# B&R Automation Studio project ABC_Pltzr
Automation Studio 4.2.4.149

## Configuration PPC70_24025GEN

### IoMap.iom - 4PPC70_101G_20W/IoMap.iom
```iecst
(*********************************************************************************
 * Copyright:
 * Author:    goran
 * Created:   August 31, 2015/10:10 PM
 *********************************************************************************
 * IO mapping
 *********************************************************************************)
VAR_CONFIG
	::gHWModules[1].ModuleOk AT %IX."X20BR9300".ModuleOk;
	::gHWModules[2].ModuleOk AT %IX."X20DI9371".ModuleOk;
	::gHWModules[3].ModuleOk AT %IX."X20DI9371a".ModuleOk;
	::gHWModules[4].ModuleOk AT %IX."X20DO4529".ModuleOk;
	::gHWModules[5].ModuleOk AT %IX."X20PS2100".ModuleOk;
	::gHWModules[6].ModuleOk AT %IX."X20DO9322".ModuleOk;
	gHWModules[7].ModuleOk AT %IX."X20DO9322a".ModuleOk;
	gHWModules[8].ModuleOk AT %IX."X20BT9400".ModuleOk;
	gHWModules[9].ModuleOk AT %IX."8I64-VFD1".ModuleOk;
	gHWModules[10].ModuleOk AT %IX."8I64-VFD2".ModuleOk;
	gHWModules[11].ModuleOk AT %IX."8I64-VFD5".ModuleOk;
	gHWModules[12].ModuleOk AT %IX."8I64-VFD52".ModuleOk;
	gHWModules[13].ModuleOk AT %IX."8I64-VFD11".ModuleOk;
	gHWModules[14].ModuleOk AT %IX."8I64-VFD12".ModuleOk;
	gHWModules[15].ModuleOk AT %IX."X67DM1321".ModuleOk;
	gHWModules[16].ModuleOk AT %IX."X67DM1321a".ModuleOk;
	gHWModules[17].ModuleOk AT %IX."X67DM1321.L08".ModuleOk;
	gHWModules[18].ModuleOk AT %IX."X67DM1321b".ModuleOk;
	::gMachineVFD[1].vfdIn.Status.ReadyToSwitchOn AT %IX."8I64-VFD1".ETAD_Input_Bool_00;
	::gMachineVFD[1].vfdIn.Status.SwitchedOn AT %IX."8I64-VFD1".ETAD_Input_Bool_01;
	::gMachineVFD[1].vfdIn.Status.OperationEnabled AT %IX."8I64-VFD1".ETAD_Input_Bool_02;
	::gMachineVFD[1].vfdIn.Status.FaultDetection AT %IX."8I64-VFD1".ETAD_Input_Bool_03;
	::gMachineVFD[1].vfdIn.Status.VoltageEnabled AT %IX."8I64-VFD1".ETAD_Input_Bool_04;
	::gMachineVFD[1].vfdIn.Status.QuickStop AT %IX."8I64-VFD1".ETAD_Input_Bool_05;
	::gMachineVFD[1].vfdIn.Status.SwitchOnDisabled AT %IX."8I64-VFD1".ETAD_Input_Bool_06;
	::gMachineVFD[1].vfdIn.Status.WarningAlarm AT %IX."8I64-VFD1".ETAD_Input_Bool_07;
	::gMachineVFD[1].vfdIn.Status.TargetReached AT %IX."8I64-VFD1".ETAD_Input_Bool_10;
	::gMachineVFD[1].vfdIn.Status.StopKey AT %IX."8I64-VFD1".ETAD_Input_Bool_14;
	::gMachineVFD[1].vfdIn.Status.Direction AT %IX."8I64-VFD1".ETAD_Input_Bool_15;
	::gMachineVFD[1].vfdIn.Status.Accelerating AT %IX."8I64-VFD1".ETI_Input_Bool_09;
	::gMachineVFD[1].vfdIn.Status.Decelerating AT %IX."8I64-VFD1".ETI_Input_Bool_10;
	::gMachineVFD[1].vfdIn.Status.FastStop AT %IX."8I64-VFD1".ETI_Input_Bool_12;
	::gMachineVFD[1].vfdIn.Status.CurrentVelocity AT %IW."8I64-VFD1".RFRD_Input;
	::gMachineVFD[1].vfdIn.Status.MotorTorque AT %IW."8I64-VFD1".OTR_Input;
	::gMachineVFD[1].vfdIn.Status.MotorCurrent AT %IW."8I64-VFD1".LCR_Input;
	::gMachineVFD[1].vfdIn.Status.DriveThermalState AT %IW."8I64-VFD1".THD_Input;
	::gMachineVFD[1].vfdIn.Status.MotorThermalState AT %IW."8I64-VFD1".THR_Input;
	::gMachineVFD[1].vfdIn.IO.LogicInput1 AT %IX."8I64-VFD1".IOLR_Input_Bool_00;
	::gMachineVFD[1].vfdIn.IO.LogicInput2 AT %IX."8I64-VFD1".IOLR_Input_Bool_01;
	::gMachineVFD[1].vfdIn.IO.LogicInput3 AT %IX."8I64-VFD1".IOLR_Input_Bool_02;
	::gMachineVFD[1].vfdIn.IO.LogicInput4 AT %IX."8I64-VFD1".IOLR_Input_Bool_03;
	::gMachineVFD[1].vfdIn.IO.Relay02State AT %IX."8I64-VFD1".IOLR_Input_Bool_09;
	::gMachineVFD[1].vfdIn.Fault.CurrentFault AT %IW."8I64-VFD1".ERRD_Input;
	::gMachineVFD[1].vfdIn.Fault.LastFault AT %IW."8I64-VFD1".LFT_Input;
	::gMachineVFD[1].vfdOut.Control.SwitchOn AT %QX."8I64-VFD1".CMDD_Output_Bool_00;
	::gMachineVFD[1].vfdOut.Control.DisableVoltage AT %QX."8I64-VFD1".CMDD_Output_Bool_01;
	::gMachineVFD[1].vfdOut.Control.QuickStop AT %QX."8I64-VFD1".CMDD_Output_Bool_02;
	::gMachineVFD[1].vfdOut.Control.EnableOperation AT %QX."8I64-VFD1".CMDD_Output_Bool_03;
	::gMachineVFD[1].vfdOut.Control.FaultReset AT %QX."8I64-VFD1".CMDD_Output_Bool_07;
	::gMachineVFD[1].vfdOut.Control.Direction AT %QX."8I64-VFD1".CMDD_Output_Bool_11;
	::gMachineVFD[1].vfdOut.Control.FastStop AT %QX."8I64-VFD1".CMDD_Output_Bool_12;
	::gMachineVFD[1].vfdOut.Control.VelocitySetpoint AT %QW."8I64-VFD1".LFRD_Output;
	::gMachineVFD[2].vfdIn.Status.ReadyToSwitchOn AT %IX."8I64-VFD2".ETAD_Input_Bool_00;
	::gMachineVFD[2].vfdIn.Status.SwitchedOn AT %IX."8I64-VFD2".ETAD_Input_Bool_01;
	::gMachineVFD[2].vfdIn.Status.OperationEnabled AT %IX."8I64-VFD2".ETAD_Input_Bool_02;
	::gMachineVFD[2].vfdIn.Status.FaultDetection AT %IX."8I64-VFD2".ETAD_Input_Bool_03;
	::gMachineVFD[2].vfdIn.Status.VoltageEnabled AT %IX."8I64-VFD2".ETAD_Input_Bool_04;
	::gMachineVFD[2].vfdIn.Status.QuickStop AT %IX."8I64-VFD2".ETAD_Input_Bool_05;
	::gMachineVFD[2].vfdIn.Status.SwitchOnDisabled AT %IX."8I64-VFD2".ETAD_Input_Bool_06;
	::gMachineVFD[2].vfdIn.Status.WarningAlarm AT %IX."8I64-VFD2".ETAD_Input_Bool_07;
	::gMachineVFD[2].vfdIn.Status.TargetReached AT %IX."8I64-VFD2".ETAD_Input_Bool_10;
	::gMachineVFD[2].vfdIn.Status.StopKey AT %IX."8I64-VFD2".ETAD_Input_Bool_14;
	::gMachineVFD[2].vfdIn.Status.Direction AT %IX."8I64-VFD2".ETAD_Input_Bool_15;
	::gMachineVFD[2].vfdIn.Status.Accelerating AT %IX."8I64-VFD2".ETI_Input_Bool_09;
	::gMachineVFD[2].vfdIn.Status.Decelerating AT %IX."8I64-VFD2".ETI_Input_Bool_10;
	::gMachineVFD[2].vfdIn.Status.FastStop AT %IX."8I64-VFD2".ETI_Input_Bool_12;
	::gMachineVFD[2].vfdIn.Status.CurrentVelocity AT %IW."8I64-VFD2".RFRD_Input;
	::gMachineVFD[2].vfdIn.Status.MotorTorque AT %IW."8I64-VFD2".OTR_Input;
	::gMachineVFD[2].vfdIn.Status.MotorCurrent AT %IW."8I64-VFD2".LCR_Input;
	::gMachineVFD[2].vfdIn.Status.DriveThermalState AT %IW."8I64-VFD2".THD_Input;
	::gMachineVFD[2].vfdIn.Status.MotorThermalState AT %IW."8I64-VFD2".THR_Input;
	::gMachineVFD[2].vfdIn.IO.LogicInput1 AT %IX."8I64-VFD2".IOLR_Input_Bool_00;
	::gMachineVFD[2].vfdIn.IO.LogicInput2 AT %IX."8I64-VFD2".IOLR_Input_Bool_01;
	::gMachineVFD[2].vfdIn.IO.LogicInput3 AT %IX."8I64-VFD2".IOLR_Input_Bool_02;
	::gMachineVFD[2].vfdIn.IO.LogicInput4 AT %IX."8I64-VFD2".IOLR_Input_Bool_03;
	::gMachineVFD[2].vfdIn.IO.Relay02State AT %IX."8I64-VFD2".IOLR_Input_Bool_09;
	::gMachineVFD[2].vfdIn.Fault.CurrentFault AT %IW."8I64-VFD2".ERRD_Input;
	::gMachineVFD[2].vfdIn.Fault.LastFault AT %IW."8I64-VFD2".LFT_Input;
	::gMachineVFD[2].vfdOut.Control.SwitchOn AT %QX."8I64-VFD2".CMDD_Output_Bool_00;
	::gMachineVFD[2].vfdOut.Control.DisableVoltage AT %QX."8I64-VFD2".CMDD_Output_Bool_01;
	::gMachineVFD[2].vfdOut.Control.QuickStop AT %QX."8I64-VFD2".CMDD_Output_Bool_02;
	::gMachineVFD[2].vfdOut.Control.EnableOperation AT %QX."8I64-VFD2".CMDD_Output_Bool_03;
	::gMachineVFD[2].vfdOut.Control.FaultReset AT %QX."8I64-VFD2".CMDD_Output_Bool_07;
	::gMachineVFD[2].vfdOut.Control.Direction AT %QX."8I64-VFD2".CMDD_Output_Bool_11;
	::gMachineVFD[2].vfdOut.Control.FastStop AT %QX."8I64-VFD2".CMDD_Output_Bool_12;
	::gMachineVFD[2].vfdOut.Control.VelocitySetpoint AT %QW."8I64-VFD2".LFRD_Output;
	gMachineVFD[5].vfdIn.Status.ReadyToSwitchOn AT %IX."8I64-VFD5".ETAD_Input_Bool_00;
	gMachineVFD[5].vfdIn.Status.SwitchedOn AT %IX."8I64-VFD5".ETAD_Input_Bool_01;
	gMachineVFD[5].vfdIn.Status.OperationEnabled AT %IX."8I64-VFD5".ETAD_Input_Bool_02;
	gMachineVFD[5].vfdIn.Status.FaultDetection AT %IX."8I64-VFD5".ETAD_Input_Bool_03;
	gMachineVFD[5].vfdIn.Status.VoltageEnabled AT %IX."8I64-VFD5".ETAD_Input_Bool_04;
	gMachineVFD[5].vfdIn.Status.QuickStop AT %IX."8I64-VFD5".ETAD_Input_Bool_05;
	gMachineVFD[5].vfdIn.Status.SwitchOnDisabled AT %IX."8I64-VFD5".ETAD_Input_Bool_06;
	gMachineVFD[5].vfdIn.Status.WarningAlarm AT %IX."8I64-VFD5".ETAD_Input_Bool_07;
	gMachineVFD[5].vfdIn.Status.TargetReached AT %IX."8I64-VFD5".ETAD_Input_Bool_10;
	gMachineVFD[5].vfdIn.Status.StopKey AT %IX."8I64-VFD5".ETAD_Input_Bool_14;
	gMachineVFD[5].vfdIn.Status.Direction AT %IX."8I64-VFD5".ETAD_Input_Bool_15;
	gMachineVFD[5].vfdIn.Status.Accelerating AT %IX."8I64-VFD5".ETI_Input_Bool_09;
	gMachineVFD[5].vfdIn.Status.Decelerating AT %IX."8I64-VFD5".ETI_Input_Bool_10;
	gMachineVFD[5].vfdIn.Status.FastStop AT %IX."8I64-VFD5".ETI_Input_Bool_12;
	gMachineVFD[5].vfdIn.Status.CurrentVelocity AT %IW."8I64-VFD5".RFRD_Input;
	gMachineVFD[5].vfdIn.Status.MotorTorque AT %IW."8I64-VFD5".OTR_Input;
	gMachineVFD[5].vfdIn.Status.MotorCurrent AT %IW."8I64-VFD5".LCR_Input;
	gMachineVFD[5].vfdIn.Status.DriveThermalState AT %IW."8I64-VFD5".THD_Input;
	gMachineVFD[5].vfdIn.Status.MotorThermalState AT %IW."8I64-VFD5".THR_Input;
	gMachineVFD[5].vfdIn.IO.LogicInput1 AT %IX."8I64-VFD5".IOLR_Input_Bool_00;
	gMachineVFD[5].vfdIn.IO.LogicInput2 AT %IX."8I64-VFD5".IOLR_Input_Bool_01;
	gMachineVFD[5].vfdIn.IO.LogicInput3 AT %IX."8I64-VFD5".IOLR_Input_Bool_02;
	gMachineVFD[5].vfdIn.IO.LogicInput4 AT %IX."8I64-VFD5".IOLR_Input_Bool_03;
	gMachineVFD[5].vfdIn.IO.Relay02State AT %IX."8I64-VFD5".IOLR_Input_Bool_09;
	gMachineVFD[5].vfdIn.Fault.CurrentFault AT %IW."8I64-VFD5".ERRD_Input;
	gMachineVFD[5].vfdIn.Fault.LastFault AT %IW."8I64-VFD5".LFT_Input;
	gMachineVFD[5].vfdOut.Control.SwitchOn AT %QX."8I64-VFD5".CMDD_Output_Bool_00;
	gMachineVFD[5].vfdOut.Control.DisableVoltage AT %QX."8I64-VFD5".CMDD_Output_Bool_01;
	gMachineVFD[5].vfdOut.Control.QuickStop AT %QX."8I64-VFD5".CMDD_Output_Bool_02;
	gMachineVFD[5].vfdOut.Control.EnableOperation AT %QX."8I64-VFD5".CMDD_Output_Bool_03;
	gMachineVFD[5].vfdOut.Control.FaultReset AT %QX."8I64-VFD5".CMDD_Output_Bool_07;
	gMachineVFD[5].vfdOut.Control.Direction AT %QX."8I64-VFD5".CMDD_Output_Bool_11;
	gMachineVFD[5].vfdOut.Control.FastStop AT %QX."8I64-VFD5".CMDD_Output_Bool_12;
	gMachineVFD[5].vfdOut.Control.VelocitySetpoint AT %QW."8I64-VFD5".LFRD_Output;
	gMachineVFD[6].vfdIn.Status.ReadyToSwitchOn AT %IX."8I64-VFD52".ETAD_Input_Bool_00;
	gMachineVFD[6].vfdIn.Status.SwitchedOn AT %IX."8I64-VFD52".ETAD_Input_Bool_01;
	gMachineVFD[6].vfdIn.Status.OperationEnabled AT %IX."8I64-VFD52".ETAD_Input_Bool_02;
	gMachineVFD[6].vfdIn.Status.FaultDetection AT %IX."8I64-VFD52".ETAD_Input_Bool_03;
	gMachineVFD[6].vfdIn.Status.VoltageEnabled AT %IX."8I64-VFD52".ETAD_Input_Bool_04;
	gMachineVFD[6].vfdIn.Status.QuickStop AT %IX."8I64-VFD52".ETAD_Input_Bool_05;
	gMachineVFD[6].vfdIn.Status.SwitchOnDisabled AT %IX."8I64-VFD52".ETAD_Input_Bool_06;
	gMachineVFD[6].vfdIn.Status.WarningAlarm AT %IX."8I64-VFD52".ETAD_Input_Bool_07;
	gMachineVFD[6].vfdIn.Status.TargetReached AT %IX."8I64-VFD52".ETAD_Input_Bool_10;
	gMachineVFD[6].vfdIn.Status.StopKey AT %IX."8I64-VFD52".ETAD_Input_Bool_14;
	gMachineVFD[6].vfdIn.Status.Direction AT %IX."8I64-VFD52".ETAD_Input_Bool_15;
	gMachineVFD[6].vfdIn.Status.Accelerating AT %IX."8I64-VFD52".ETI_Input_Bool_09;
	gMachineVFD[6].vfdIn.Status.Decelerating AT %IX."8I64-VFD52".ETI_Input_Bool_10;
	gMachineVFD[6].vfdIn.Status.FastStop AT %IX."8I64-VFD52".ETI_Input_Bool_12;
	gMachineVFD[6].vfdIn.Status.CurrentVelocity AT %IW."8I64-VFD52".RFRD_Input;
	gMachineVFD[6].vfdIn.Status.MotorTorque AT %IW."8I64-VFD52".OTR_Input;
	gMachineVFD[6].vfdIn.Status.MotorCurrent AT %IW."8I64-VFD52".LCR_Input;
	gMachineVFD[6].vfdIn.Status.DriveThermalState AT %IW."8I64-VFD52".THD_Input;
	gMachineVFD[6].vfdIn.Status.MotorThermalState AT %IW."8I64-VFD52".THR_Input;
	gMachineVFD[6].vfdIn.IO.LogicInput1 AT %IX."8I64-VFD52".IOLR_Input_Bool_00;
	gMachineVFD[6].vfdIn.IO.LogicInput2 AT %IX."8I64-VFD52".IOLR_Input_Bool_01;
	gMachineVFD[6].vfdIn.IO.LogicInput3 AT %IX."8I64-VFD52".IOLR_Input_Bool_02;
	gMachineVFD[6].vfdIn.IO.LogicInput4 AT %IX."8I64-VFD52".IOLR_Input_Bool_03;
	gMachineVFD[6].vfdIn.IO.Relay02State AT %IX."8I64-VFD52".IOLR_Input_Bool_09;
	gMachineVFD[6].vfdIn.Fault.CurrentFault AT %IW."8I64-VFD52".ERRD_Input;
	gMachineVFD[6].vfdIn.Fault.LastFault AT %IW."8I64-VFD52".LFT_Input;
	gMachineVFD[6].vfdOut.Control.SwitchOn AT %QX."8I64-VFD52".CMDD_Output_Bool_00;
	gMachineVFD[6].vfdOut.Control.DisableVoltage AT %QX."8I64-VFD52".CMDD_Output_Bool_01;
	gMachineVFD[6].vfdOut.Control.QuickStop AT %QX."8I64-VFD52".CMDD_Output_Bool_02;
	gMachineVFD[6].vfdOut.Control.EnableOperation AT %QX."8I64-VFD52".CMDD_Output_Bool_03;
	gMachineVFD[6].vfdOut.Control.FaultReset AT %QX."8I64-VFD52".CMDD_Output_Bool_07;
	gMachineVFD[6].vfdOut.Control.Direction AT %QX."8I64-VFD52".CMDD_Output_Bool_11;
	gMachineVFD[6].vfdOut.Control.FastStop AT %QX."8I64-VFD52".CMDD_Output_Bool_12;
	gMachineVFD[6].vfdOut.Control.VelocitySetpoint AT %QW."8I64-VFD52".LFRD_Output;
	gMachineVFD[11].vfdIn.Status.ReadyToSwitchOn AT %IX."8I64-VFD11".ETAD_Input_Bool_00;
	gMachineVFD[11].vfdIn.Status.SwitchedOn AT %IX."8I64-VFD11".ETAD_Input_Bool_01;
	gMachineVFD[11].vfdIn.Status.OperationEnabled AT %IX."8I64-VFD11".ETAD_Input_Bool_02;
	gMachineVFD[11].vfdIn.Status.FaultDetection AT %IX."8I64-VFD11".ETAD_Input_Bool_03;
	gMachineVFD[11].vfdIn.Status.VoltageEnabled AT %IX."8I64-VFD11".ETAD_Input_Bool_04;
	gMachineVFD[11].vfdIn.Status.QuickStop AT %IX."8I64-VFD11".ETAD_Input_Bool_05;
	gMachineVFD[11].vfdIn.Status.SwitchOnDisabled AT %IX."8I64-VFD11".ETAD_Input_Bool_06;
	gMachineVFD[11].vfdIn.Status.WarningAlarm AT %IX."8I64-VFD11".ETAD_Input_Bool_07;
	gMachineVFD[11].vfdIn.Status.TargetReached AT %IX."8I64-VFD11".ETAD_Input_Bool_10;
	gMachineVFD[11].vfdIn.Status.StopKey AT %IX."8I64-VFD11".ETAD_Input_Bool_14;
	gMachineVFD[11].vfdIn.Status.Direction AT %IX."8I64-VFD11".ETAD_Input_Bool_15;
	gMachineVFD[11].vfdIn.Status.Accelerating AT %IX."8I64-VFD11".ETI_Input_Bool_09;
	gMachineVFD[11].vfdIn.Status.Decelerating AT %IX."8I64-VFD11".ETI_Input_Bool_10;
	gMachineVFD[11].vfdIn.Status.FastStop AT %IX."8I64-VFD11".ETI_Input_Bool_12;
	gMachineVFD[11].vfdIn.Status.CurrentVelocity AT %IW."8I64-VFD11".RFRD_Input;
	gMachineVFD[11].vfdIn.Status.MotorTorque AT %IW."8I64-VFD11".OTR_Input;
	gMachineVFD[11].vfdIn.Status.MotorCurrent AT %IW."8I64-VFD11".LCR_Input;
	gMachineVFD[11].vfdIn.Status.DriveThermalState AT %IW."8I64-VFD11".THD_Input;
	gMachineVFD[11].vfdIn.Status.MotorThermalState AT %IW."8I64-VFD11".THR_Input;
	gMachineVFD[11].vfdIn.IO.LogicInput1 AT %IX."8I64-VFD11".IOLR_Input_Bool_00;
	gMachineVFD[11].vfdIn.IO.LogicInput2 AT %IX."8I64-VFD11".IOLR_Input_Bool_01;
	gMachineVFD[11].vfdIn.IO.LogicInput3 AT %IX."8I64-VFD11".IOLR_Input_Bool_02;
	gMachineVFD[11].vfdIn.IO.LogicInput4 AT %IX."8I64-VFD11".IOLR_Input_Bool_03;
	gMachineVFD[11].vfdIn.IO.Relay02State AT %IX."8I64-VFD11".IOLR_Input_Bool_09;
	gMachineVFD[11].vfdIn.Fault.CurrentFault AT %IW."8I64-VFD11".ERRD_Input;
	gMachineVFD[11].vfdIn.Fault.LastFault AT %IW."8I64-VFD11".LFT_Input;
	gMachineVFD[11].vfdOut.Control.SwitchOn AT %QX."8I64-VFD11".CMDD_Output_Bool_00;
	gMachineVFD[11].vfdOut.Control.DisableVoltage AT %QX."8I64-VFD11".CMDD_Output_Bool_01;
	gMachineVFD[11].vfdOut.Control.QuickStop AT %QX."8I64-VFD11".CMDD_Output_Bool_02;
	gMachineVFD[11].vfdOut.Control.EnableOperation AT %QX."8I64-VFD11".CMDD_Output_Bool_03;
	gMachineVFD[11].vfdOut.Control.FaultReset AT %QX."8I64-VFD11".CMDD_Output_Bool_07;
	gMachineVFD[11].vfdOut.Control.Direction AT %QX."8I64-VFD11".CMDD_Output_Bool_11;
	gMachineVFD[11].vfdOut.Control.FastStop AT %QX."8I64-VFD11".CMDD_Output_Bool_12;
	gMachineVFD[11].vfdOut.Control.VelocitySetpoint AT %QW."8I64-VFD11".LFRD_Output;
	gMachineVFD[12].vfdIn.Status.ReadyToSwitchOn AT %IX."8I64-VFD12".ETAD_Input_Bool_00;
	gMachineVFD[12].vfdIn.Status.SwitchedOn AT %IX."8I64-VFD12".ETAD_Input_Bool_01;
	gMachineVFD[12].vfdIn.Status.OperationEnabled AT %IX."8I64-VFD12".ETAD_Input_Bool_02;
	gMachineVFD[12].vfdIn.Status.FaultDetection AT %IX."8I64-VFD12".ETAD_Input_Bool_03;
	gMachineVFD[12].vfdIn.Status.VoltageEnabled AT %IX."8I64-VFD12".ETAD_Input_Bool_04;
	gMachineVFD[12].vfdIn.Status.QuickStop AT %IX."8I64-VFD12".ETAD_Input_Bool_05;
	gMachineVFD[12].vfdIn.Status.SwitchOnDisabled AT %IX."8I64-VFD12".ETAD_Input_Bool_06;
	gMachineVFD[12].vfdIn.Status.WarningAlarm AT %IX."8I64-VFD12".ETAD_Input_Bool_07;
	gMachineVFD[12].vfdIn.Status.TargetReached AT %IX."8I64-VFD12".ETAD_Input_Bool_10;
	gMachineVFD[12].vfdIn.Status.StopKey AT %IX."8I64-VFD12".ETAD_Input_Bool_14;
	gMachineVFD[12].vfdIn.Status.Direction AT %IX."8I64-VFD12".ETAD_Input_Bool_15;
	gMachineVFD[12].vfdIn.Status.Accelerating AT %IX."8I64-VFD12".ETI_Input_Bool_09;
	gMachineVFD[12].vfdIn.Status.Decelerating AT %IX."8I64-VFD12".ETI_Input_Bool_10;
	gMachineVFD[12].vfdIn.Status.FastStop AT %IX."8I64-VFD12".ETI_Input_Bool_12;
	gMachineVFD[12].vfdIn.Status.CurrentVelocity AT %IW."8I64-VFD12".RFRD_Input;
	gMachineVFD[12].vfdIn.Status.MotorTorque AT %IW."8I64-VFD12".OTR_Input;
	gMachineVFD[12].vfdIn.Status.MotorCurrent AT %IW."8I64-VFD12".LCR_Input;
	gMachineVFD[12].vfdIn.Status.DriveThermalState AT %IW."8I64-VFD12".THD_Input;
	gMachineVFD[12].vfdIn.Status.MotorThermalState AT %IW."8I64-VFD12".THR_Input;
	gMachineVFD[12].vfdIn.IO.LogicInput1 AT %IX."8I64-VFD12".IOLR_Input_Bool_00;
	gMachineVFD[12].vfdIn.IO.LogicInput2 AT %IX."8I64-VFD12".IOLR_Input_Bool_01;
	gMachineVFD[12].vfdIn.IO.LogicInput3 AT %IX."8I64-VFD12".IOLR_Input_Bool_02;
	gMachineVFD[12].vfdIn.IO.LogicInput4 AT %IX."8I64-VFD12".IOLR_Input_Bool_03;
	gMachineVFD[12].vfdIn.IO.Relay02State AT %IX."8I64-VFD12".IOLR_Input_Bool_09;
	gMachineVFD[12].vfdIn.Fault.CurrentFault AT %IW."8I64-VFD12".ERRD_Input;
	gMachineVFD[12].vfdIn.Fault.LastFault AT %IW."8I64-VFD12".LFT_Input;
	gMachineVFD[12].vfdOut.Control.SwitchOn AT %QX."8I64-VFD12".CMDD_Output_Bool_00;
	gMachineVFD[12].vfdOut.Control.DisableVoltage AT %QX."8I64-VFD12".CMDD_Output_Bool_01;
	gMachineVFD[12].vfdOut.Control.QuickStop AT %QX."8I64-VFD12".CMDD_Output_Bool_02;
	gMachineVFD[12].vfdOut.Control.EnableOperation AT %QX."8I64-VFD12".CMDD_Output_Bool_03;
	gMachineVFD[12].vfdOut.Control.FaultReset AT %QX."8I64-VFD12".CMDD_Output_Bool_07;
	gMachineVFD[12].vfdOut.Control.Direction AT %QX."8I64-VFD12".CMDD_Output_Bool_11;
	gMachineVFD[12].vfdOut.Control.FastStop AT %QX."8I64-VFD12".CMDD_Output_Bool_12;
	gMachineVFD[12].vfdOut.Control.VelocitySetpoint AT %QW."8I64-VFD12".LFRD_Output;
	::gMachineIO.din.Guard_DS1 AT %IX."X20DI9371".DigitalInput01;
	::gMachineIO.din.Guard_DS2 AT %IX."X20DI9371".DigitalInput02;
	::gMachineIO.din.Guard_DS3 AT %IX."X20DI9371".DigitalInput03;
	::gMachineIO.din.EStop_PB1 AT %IX."X20DI9371".DigitalInput07;
	::gMachineIO.din.EStop_PB2 AT %IX."X20DI9371".DigitalInput08;
	::gMachineIO.din.EStop_PB3 AT %IX."X20DI9371".DigitalInput09;
	::gMachineIO.din.EStop_PB4 AT %IX."X20DI9371".DigitalInput10;
	::gMachineIO.din.MotorOverloads_OL AT %IX."X20DI9371a".DigitalInput01;
	::gMachineIO.din.MCR AT %IX."X20DI9371a".DigitalInput02;
	::gMachineIO.din.CustomerDischargeEnable_CR6 AT %IX."X20DI9371a".DigitalInput03;
	gMachineIO.din.PalleteDischLightCurtain_OSSD1 AT %IX."X20DI9371a".DigitalInput04;
	gMachineIO.din.PalleteDischLightCurtain_OSSD2 AT %IX."X20DI9371a".DigitalInput05;
	gMachineIO.din.AirPressureSwitch_APS AT %IX."X20DI9371a".DigitalInput06;
	::gMachineIO.dout.MachineFaultBeacon_LT1 AT %QX."X20DO4529".DigitalOutput01;
	::gMachineIO.dout.MachineOkBeacon_LT2 AT %QX."X20DO4529".DigitalOutput02;
	::gMachineIO.dout.PalletLowSupplyBeacon_LT3 AT %QX."X20DO4529".DigitalOutput03;
	::gMachineIO.dout.CustomerMachineRunning_CR5 AT %QX."X20DO4529".DigitalOutput04;
	::gMachineIO.dout.LayerStopBarRaise_M3F AT %QX."X20DO9322".DigitalOutput03;
	::gMachineIO.dout.LayerStopBarLower_M3R AT %QX."X20DO9322".DigitalOutput04;
	::gMachineIO.dout.RowFormingRollers_M5 AT %QX."X20DO9322".DigitalOutput07;
	::gMachineIO.dout.ProductInfeedCV_M6 AT %QX."X20DO9322".DigitalOutput08;
	::gMachineIO.dout.PalletDispenserCV_M7 AT %QX."X20DO9322".DigitalOutput09;
	::gMachineIO.dout.PalletDispenserRaise_M8F AT %QX."X20DO9322".DigitalOutput10;
	::gMachineIO.dout.PalletDispenserLower_M8R AT %QX."X20DO9322".DigitalOutput11;
	::gMachineIO.dout.CustomerMachineRunning_CR4 AT %QX."X20DO9322".DigitalOutput12;
	::gMachineIO.din.ElevatorDetectPalletLayerLF_EE1 AT %IX."X67DM1321".DigitalInput01;
	::gMachineIO.din.ElevatorChainSlackLF_LS7 AT %IX."X67DM1321".DigitalInput03;
	::gMachineIO.din.ElevatorChainSlackRT_LS8 AT %IX."X67DM1321".DigitalInput04;
	::gMachineIO.din.TransferTableAtPallete_PR5 AT %IX."X67DM1321".DigitalInput05;
	::gMachineIO.din.TransferTableAtGrouping_PR6 AT %IX."X67DM1321".DigitalInput06;
	::gMachineIO.din.LayerStopBarUp_PR7 AT %IX."X67DM1321".DigitalInput07;
	::gMachineIO.din.LayerStopBarDown_PR8 AT %IX."X67DM1321".DigitalInput08;
	::gMachineIO.dout.SideSquaringExtend_SOL8A AT %QX."X67DM1321a".DigitalOutput01;
	::gMachineIO.dout.SideSquaringRetract_SOL8B AT %QX."X67DM1321a".DigitalOutput02;
	::gMachineIO.dout.CaseTurnerRaise_SOL2A AT %QX."X67DM1321.L08".DigitalOutput01;
	::gMachineIO.dout.CaseTurnerLower_SOL2B AT %QX."X67DM1321.L08".DigitalOutput02;
	::gMachineIO.dout.BladeStop1Up_SOL3A AT %QX."X67DM1321.L08".DigitalOutput03;
	::gMachineIO.dout.BladeStop1Dw_SOL3B AT %QX."X67DM1321.L08".DigitalOutput04;
	::gMachineIO.din.ProductAtInfeed_EE2Phy AT %IX."X67DM1321.L08".DigitalInput13;
	::gMachineIO.din.RowTooLong_EE8Phy AT %IX."X67DM1321.L08".DigitalInput14;
	::gMachineIO.din.RowPusherReturned_PR11 AT %IX."X67DM1321.L08".DigitalInput15;
	::gMachineIO.din.RowPusherAtElevator_PR13 AT %IX."X67DM1321.L08".DigitalInput16;
	::gMachineIO.din.ElevatorFullUp_PR1 AT %IX."X67DM1321b".DigitalInput01;
	::gMachineIO.din.ElevatorFullDown_PR2 AT %IX."X67DM1321b".DigitalInput02;
	::gMachineIO.din.ElevatorAtGroupingLower_PR3 AT %IX."X67DM1321b".DigitalInput03;
	::gMachineIO.din.ElevatorAtGroupingRaise_PR4 AT %IX."X67DM1321b".DigitalInput04;
	::gMachineIO.din.ElevatorStopBlockLF_PR33 AT %IX."X67DM1321b".DigitalInput05;
	::gMachineIO.din.ElevatorStopBlockRT_PR34 AT %IX."X67DM1321b".DigitalInput06;
	::gMachineIO.din.PalletAtMachine_EE12 AT %IX."X67DM1321b".DigitalInput07;
	::gMachineIO.din.PalletAtDischarge_EE16 AT %IX."X67DM1321b".DigitalInput08;
	::gMachineIO.dout.AirDump_SOL0 AT %QX."X20DO9322a".DigitalOutput01;
	::gMachineIO.dout.SheetInserterToMagazine AT %QX."X20DO9322a".DigitalOutput02;
	gMachineIO.din.PalletMagazineControl_SS2 AT %IX."X20DI9371a".DigitalInput07;
	gMachineIO.dout.BladeStop2Up_SOL4A AT %QX."X67DM1321.L08".DigitalOutput05;
	gMachineIO.dout.BladeStop3Up_SOL5A AT %QX."X67DM1321.L08".DigitalOutput07;
	gMachineIO.dout.BladeStop4Up_SOL6A AT %QX."X67DM1321.L08".DigitalOutput09;
	gMachineIO.dout.BladeStop5Up_SOL13A AT %QX."X67DM1321.L08".DigitalOutput11;
	gMachineIO.dout.BladeStop2Dw_SOL4B AT %QX."X67DM1321.L08".DigitalOutput06;
	gMachineIO.dout.BladeStop3Dw_SOL5B AT %QX."X67DM1321.L08".DigitalOutput08;
	gMachineIO.dout.BladeStop4Dw_SOL6B AT %QX."X67DM1321.L08".DigitalOutput10;
	gMachineIO.dout.BladeStop5Dw_SOL13B AT %QX."X67DM1321.L08".DigitalOutput12;
	gMachineIO.dout.RowPusherForward_M4F AT %QX."X20DO9322".DigitalOutput05;
	gMachineIO.dout.RowPusherReturn_M4R AT %QX."X20DO9322".DigitalOutput06;
	gMachineIO.dout.FrontSquaringExtend_SOL11A AT %QX."X67DM1321a".DigitalOutput03;
	gMachineIO.dout.FrontSquaringRetract_SOL11B AT %QX."X67DM1321a".DigitalOutput04;
	gMachineIO.dout.BladeStop6Up_SOL14A AT %QX."X67DM1321c".DigitalOutput01;
	::gMachineIO.dout.BladeStop6Dw_SOL14B AT %QX."X67DM1321c".DigitalOutput02;
	gMachineIO.din.Guard_DS4 AT %IX."X20DI9371".DigitalInput04;
	gMachineIO.din.Guard_DS5 AT %IX."X20DI9371".DigitalInput05;
	::gMachineIO.din.ProductAtStage_EE4Phy AT %IX."X67DM1321c".DigitalInput03;
END_VAR
```


## Logical view

Binary libraries used (declarations not repeated): AsARCfg, AsIOAcc, asstring, AsUDP, Visapi

### MachineIO.var
```iecst
(*********************************************************************************
 * Copyright: Piedmont Automation Inc
 * Author:    Goran
 * Created:   Jun 26, 2015/11:38 AM
 *********************************************************************************
 * Declaration of global variables
 *********************************************************************************)
VAR
	gHWModules : ARRAY[0..APP_HWMODULE_IDXLAST] OF paiBnRHWModuleInfo_typ;
	gMachineIO : machineIO_typ := (0);
END_VAR
```

- caseCmdEditorItems.clm (not shown)

- Button.fninfo (not shown)

- Header.fninfo (not shown)

- Status.fninfo (not shown)

- TabButtonText.fninfo (not shown)

- paiHmiTabs7.layer (not shown)

- paiHmiTabs9.layer (not shown)

- paiMpRecipeUIXML.layer (not shown)

- MpAlphaPad.tpr (not shown)

### dvframe.typ
```iecst
(********************************************************************
 * COPYRIGHT (C) BERNECKER + RAINER, AUSTRIA, A-5142 EGGELSBERG
 ********************************************************************
 * Library: DVFrame
 * File: DVFrame.typ
 * Created: 11.11.2003
 ********************************************************************
 * Global data types of library DVFrame
 ********************************************************************)
TYPE
	XOPENCONFIG : STRUCT
		idle	: UINT ;					(*maximum idle time between characters*)
		delimc	: UINT ;					(*activate the frame delimiters, standard value : 0*)
		delim	: ARRAY[0..1] OF USINT ;	(*frame delimiters, default value: 0,0*)
		tx_cnt	: UINT ;					(*number of send buffers (maximum 8), default value: 2*)
		rx_cnt	: UINT ;					(*number of receive buffers (maximum 8), default value: 2*)
		tx_len	: UINT ;					(*send buffer length, default value: 256 bytes*)
		rx_len	: UINT ;					(*receive buffer length, default value: 256 bytes*)
		argc	: UINT ;					(*number of additional arguments in argv, default value: 0*)
		argv	: UDINT ;					(*address for a UDINT field with additional arguments, default value: 0*)
	END_STRUCT;
END_TYPE
```

### EthSock.typ
```iecst
(********************************************************************
 * COPYRIGHT (C) BERNECKER + RAINER, AUSTRIA, A-5142 EGGELSBERG
 ********************************************************************
 * Library: EthSock
 * File: EthSock.typ
 * Created: 11.11.2003
 ********************************************************************
 * Global data types of library EthSock
 ********************************************************************)
TYPE
	ETH_timeval_typ : STRUCT
		tv_sec	: DINT ;
		tv_usec	: DINT ;
	END_STRUCT;
	ETH_fd_set_typ : STRUCT
		fds_bits	: ARRAY[0..7] OF DINT ;
	END_STRUCT;
	ETH_sockaddr_typ : STRUCT
		sin_family	: UINT ;
		sin_port	: UINT ;
		sin_addr	: UDINT ;
		sin_zero	: ARRAY[0..7] OF USINT ;
	END_STRUCT;
END_TYPE
```

### Program Logical/MachineControl/appHmi (ANSIC)

#### paiHmiAlert.c
```c
/********************************************************************
 * COPYRIGHT -- pai
 ********************************************************************
 * Program: hmilogic
 * File: hmiAlert.c
 * Author: goran
 * Created: September 05, 2013
 *******************************************************************/

#include <bur/plctypes.h>
#ifdef _DEFAULT_INCLUDES
	#include <AsDefault.h>
#endif

/**
Bit manipulaiton utility functions.
 */
#include "../bglib/bgBitUtilities.h"

/**
String manipulaiton utility functions.
 */
//#include <../../bglib/bgsprintf.h>
#include "../bglib/bgstring.h"

/**
 Timer control utility functions.
 */
//#include <../../bglib/bgTimer1ms.h>

//Control on/off a variable that control the visibility of the alarm alert display
void paiHmiAlertHide(paiHmiAlert_typ* p)
{
	//control visibility of the layer > make it invisible
	bgBitSetUINT(&p->status, 0, 1);
}

// Is alert message active (visible)?
BOOL paiHmiAlertIsActive(paiHmiAlert_typ* p)
{
	if(bgTimerIsTimeOut(&p->tmr1))
		return 0;
	else
		return 1;
}

// Show the alert with a specified text and for a selected amount of time
void paiHmiAlertShow(paiHmiAlert_typ* p, char* headerText, char* alertText, UDINT alertDuration)
{
	if(!p)
		return;

	//control visibility of the layer > make it visible
	bgBitSetUINT(&p->status, 0, 0);

	if(!headerText){
		bgStrCpyN(p->header, "Message", sizeof(p->header));
	}else{
		bgStrCpyN(p->header, headerText, sizeof(p->header));
	}

	if(!p->message){
		bgStrCpyN(p->message, "No message.", sizeof(p->message));
	}else{
		bgStrCpyN(p->message, alertText, sizeof(p->message));
	}
	if(alertDuration < 500){
		alertDuration = 500;
	}else
	if(alertDuration > 10000){
		alertDuration = 10000;
	}
	bgTimerStart(&p->tmr1, alertDuration);
}

// Cyclic operation of the alert box.
void paiHmiAlertCyclic(paiHmiAlert_typ* p)
{
	bgTimerCyclic(&p->tmr1);
	if( !(p->status & 0x1) && bgTimerIsTimeOut(&p->tmr1) ){
		paiHmiAlertHide(p);
	}
}
//eof
```

### Program Logical/MachineControl/drycypal

#### Cyclic.st
```iecst
PROGRAM _CYCLIC
	(* Insert code here *)
	palleteTimer();

	IF ((dryCycleStatePallete <> 0) AND (NOT gCtrl.main.noFaults)) THEN
		dryCycleStatePallete := 0;
	END_IF;

	CASE dryCycleStatePallete OF
		0 : IF gCtrl.main.modeAuto THEN//wait here for auto mode
				dryCycleStatePallete := 10;
				gCtrl.palletDispenser.hmiBtnClawsLiftToTop := 1;
//				elevatorTimer.IN := 0;
//				elevatorTimer.PT := T#3s * gCtrlAnimation.currentLayer;
			END_IF;
		10: //make sure to start at top
			IF gCtrl.palletDispenser.atTop THEN
				gCtrl.palletDispenser.hmiBtnPalletClawsOpenClose := 1;//CLOSE CLAWS
			END_IF;
			IF gCtrl.palletDispenser.atTop AND gCtrl.palletDispenser.hmiBtnPalletClawsOpenClose THEN
				gCtrl.palletDispenser.hmiBtnClawsLiftToBottom := 1;//GO TO BOTTOM
				dryCycleStatePallete := 20;
			END_IF;
		20://wait to bottom
			IF gCtrl.palletDispenser.atBottom THEN//WAIT TO GET TO BOTTOM
				gCtrl.palletDispenser.hmiBtnPalletClawsOpenClose := 0;//OPEN CLAWS
				palleteTimer.IN := 0;
				palleteTimer.PT := T#3s;
				dryCycleStatePallete := 30;
			END_IF;
		30://WAIT FOR CLAWS TO OPEN
			palleteTimer.IN := 1;
			IF palleteTimer.Q THEN
				gCtrl.palletDispenser.hmiBtnClawsLiftToMidLo := 1;//move to MID low
				dryCycleStatePallete := 40;
			END_IF;
		40:
			IF gCtrl.palletDispenser.atMidLo THEN//Wait for At mit Low
				gCtrl.palletDispenser.hmiBtnPalletClawsOpenClose := 1;//CLOSE CLAWS
				palleteTimer.IN := 0;
				palleteTimer.PT := T#3s;
				dryCycleStatePallete := 50;
			END_IF;

		50://
			palleteTimer.IN := 1;
			IF palleteTimer.Q THEN
				gCtrl.palletDispenser.hmiBtnClawsLiftToTop := 1;
				dryCycleStatePallete := 60;
			END_IF;
		60://wait for elevator to come back home
			IF gCtrl.palletDispenser.atTop THEN
				palleteTimer.IN := 0;
				palleteTimer.PT := T#10s;
				dryCycleStatePallete := 70;
			END_IF;
		70://dwell here
			palleteTimer.IN := 1;
			IF palleteTimer.Q THEN
				dryCycleStatePallete := 80;
				gCtrl.palletDispenser.hmiBtnClawsLiftToMidLo := 1;
			END_IF;

		80:
			IF gCtrl.palletDispenser.atMidLo THEN//Wait for At mit Low
				gCtrl.palletDispenser.hmiBtnPalletClawsOpenClose := 0;//OPEN CLAWS
				palleteTimer.IN := 0;
				palleteTimer.PT := T#3s;
				dryCycleStatePallete := 90;
			END_IF;
		90:
			palleteTimer.IN := 1;
			IF palleteTimer.Q THEN
				gCtrl.palletDispenser.hmiBtnClawsLiftToBottom := 1;
				dryCycleStatePallete := 100;
			END_IF;
		100:
			IF gCtrl.palletDispenser.atBottom THEN//Wait for At mit Low
				gCtrl.palletDispenser.hmiBtnPalletClawsOpenClose := 1;//CLOSE CLAWS
				palleteTimer.IN := 0;
				palleteTimer.PT := T#3s;
				dryCycleStatePallete := 110;
			END_IF;

		110:
			palleteTimer.IN := 1;
			IF palleteTimer.Q THEN
				gCtrl.palletDispenser.hmiBtnClawsLiftToTop := 1;
				dryCycleStatePallete := 120;
			END_IF;

		120:
			IF gCtrl.palletDispenser.atTop THEN
				palleteTimer.IN := 0;
				palleteTimer.PT := T#15s;
				dryCycleStatePallete := 130;
			END_IF;
		130:
			palleteTimer.IN := 1;
			IF palleteTimer.Q THEN
				dryCycleStatePallete := 0;
			END_IF;
		ELSE

	END_CASE;

END_PROGRAM
```

### Program Logical/MachineControl/palletinfdis

#### Cyclic.ld
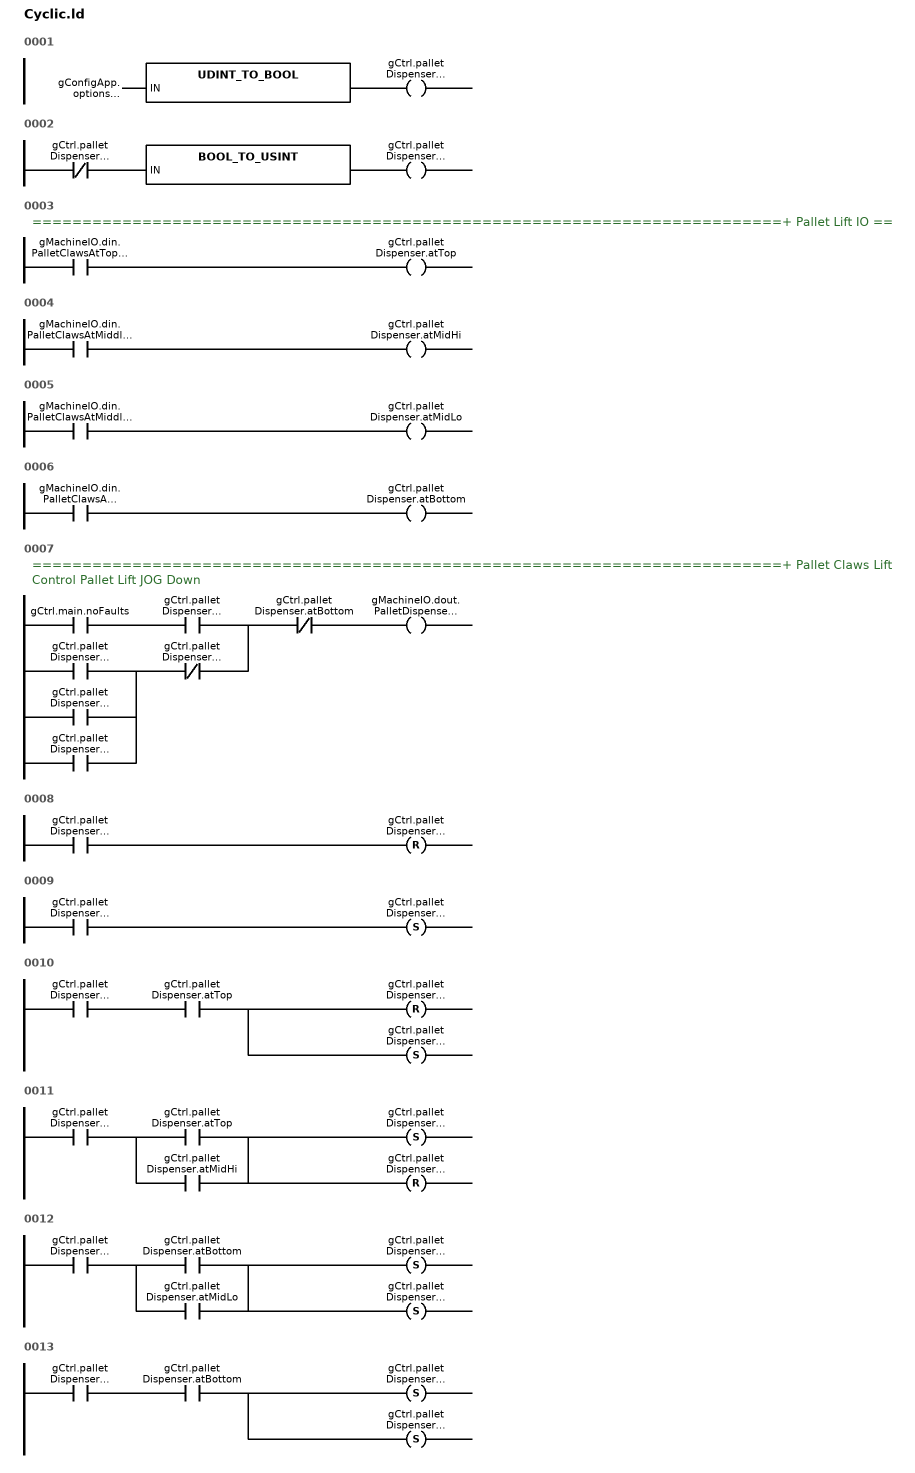
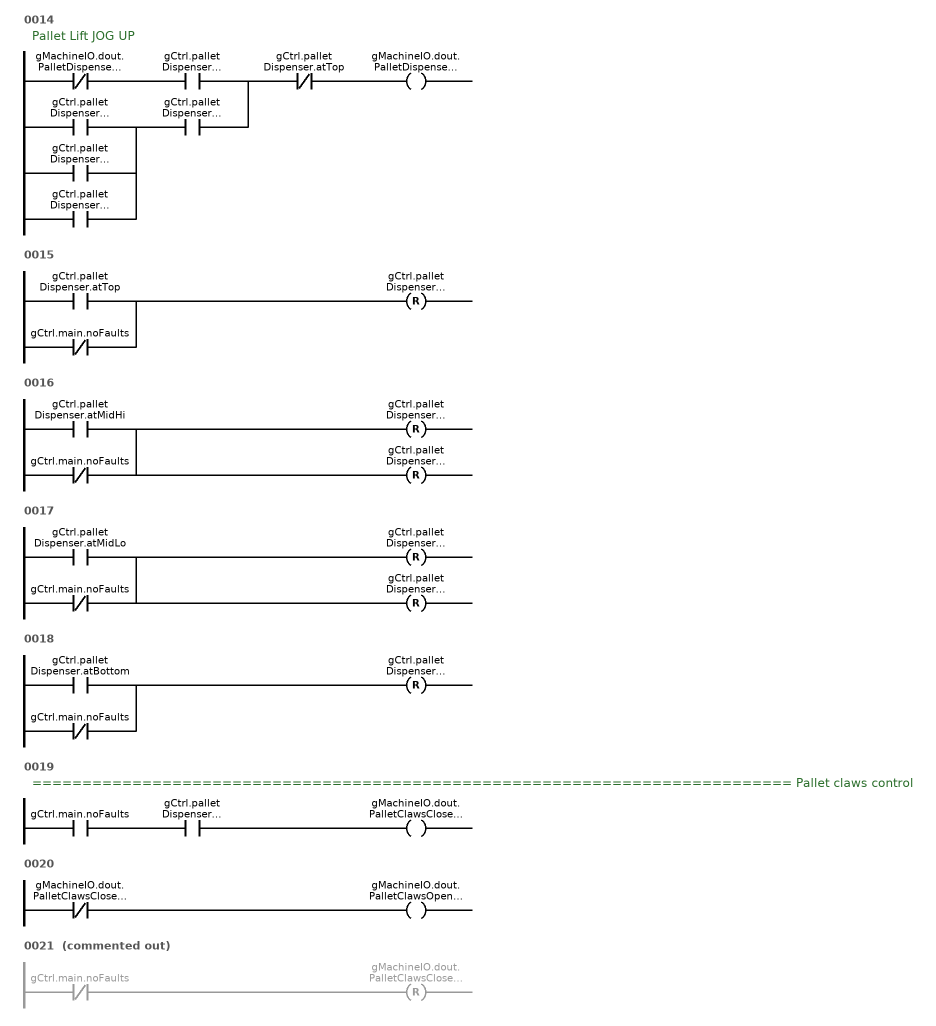
Ladder, written as Structured Text:
```iecst
PROGRAM _CYCLIC
VAR
    _p1 : BOOL;
    _p2 : BOOL;
    _p3 : BOOL;
    _p4 : BOOL;
    _p5 : BOOL;
    _p6 : BOOL;
    _p7 : BOOL;
    _p8 : BOOL;
    _p9 : BOOL;
    _p10 : BOOL;
END_VAR
(* Network 1 *)
gCtrl.palletDispenser.palletDispenserEquipped := UDINT_TO_BOOL(gConfigApp.options.palletDispenserOption);

(* Network 2 *)
gCtrl.palletDispenser.palletDispenserEquippedVis := BOOL_TO_USINT(NOT gCtrl.palletDispenser.palletDispenserEquipped);

(* Network 3: ===========================================================================+ Pallet Lift IO == *)
gCtrl.palletDispenser.atTop := gMachineIO.din.PalletClawsAtTop_PR14;

(* Network 4 *)
gCtrl.palletDispenser.atMidHi := gMachineIO.din.PalletClawsAtMiddleHi_PR15A;

(* Network 5 *)
gCtrl.palletDispenser.atMidLo := gMachineIO.din.PalletClawsAtMiddleLow_PR15;

(* Network 6 *)
gCtrl.palletDispenser.atBottom := gMachineIO.din.PalletClawsAtBottom_PR16;

(* Network 7: ===========================================================================+ Pallet Claws Lift Control Pallet Lift JOG Down   *)
gMachineIO.dout.PalletDispenserLower_M8R := ((gCtrl.main.noFaults AND gCtrl.palletDispenser.hmiBtnClawsLiftDwJog) OR ((gCtrl.palletDispenser.hmiBtnClawsLiftToBottom OR gCtrl.palletDispenser.flagClawsLiftToMidHi OR gCtrl.palletDispenser.flagClawsLiftToMidLo) AND NOT gCtrl.palletDispenser.flagMoveUp)) AND NOT gCtrl.palletDispenser.atBottom;

(* Network 8 *)
IF gCtrl.palletDispenser.hmiBtnClawsLiftToBottom THEN gCtrl.palletDispenser.flagMoveUp := FALSE; END_IF;

(* Network 9 *)
IF gCtrl.palletDispenser.hmiBtnClawsLiftToTop THEN gCtrl.palletDispenser.flagMoveUp := TRUE; END_IF;

(* Network 10 *)
_p1 := gCtrl.palletDispenser.hmiBtnClawsLiftToMidHi AND gCtrl.palletDispenser.atTop;
IF _p1 THEN
    gCtrl.palletDispenser.flagMoveUp := FALSE;
    gCtrl.palletDispenser.flagClawsLiftToMidHi := TRUE;
END_IF;

(* Network 11 *)
_p2 := gCtrl.palletDispenser.hmiBtnClawsLiftToMidLo AND gCtrl.palletDispenser.atTop;
_p3 := gCtrl.palletDispenser.hmiBtnClawsLiftToMidLo AND gCtrl.palletDispenser.atMidHi;
IF _p2 OR _p3 THEN
    gCtrl.palletDispenser.flagClawsLiftToMidLo := TRUE;
    gCtrl.palletDispenser.flagMoveUp := FALSE;
END_IF;

(* Network 12 *)
_p4 := gCtrl.palletDispenser.hmiBtnClawsLiftToMidHi AND gCtrl.palletDispenser.atBottom;
_p5 := gCtrl.palletDispenser.hmiBtnClawsLiftToMidHi AND gCtrl.palletDispenser.atMidLo;
IF _p4 OR _p5 THEN
    gCtrl.palletDispenser.flagMoveUp := TRUE;
    gCtrl.palletDispenser.flagClawsLiftToMidHi := TRUE;
END_IF;

(* Network 13 *)
_p6 := gCtrl.palletDispenser.hmiBtnClawsLiftToMidLo AND gCtrl.palletDispenser.atBottom;
IF _p6 THEN
    gCtrl.palletDispenser.flagClawsLiftToMidLo := TRUE;
    gCtrl.palletDispenser.flagMoveUp := TRUE;
END_IF;

(* Network 14: Pallet Lift JOG UP *)
gMachineIO.dout.PalletDispenserRaise_M8F := ((NOT gMachineIO.dout.PalletDispenserLower_M8R AND gCtrl.palletDispenser.hmiBtnClawsLiftUpJog) OR ((gCtrl.palletDispenser.hmiBtnClawsLiftToTop OR gCtrl.palletDispenser.flagClawsLiftToMidLo OR gCtrl.palletDispenser.flagClawsLiftToMidHi) AND gCtrl.palletDispenser.flagMoveUp)) AND NOT gCtrl.palletDispenser.atTop;

(* Network 15 *)
IF gCtrl.palletDispenser.atTop OR NOT gCtrl.main.noFaults THEN
    gCtrl.palletDispenser.hmiBtnClawsLiftToTop := FALSE;
END_IF;

(* Network 16 *)
_p7 := gCtrl.palletDispenser.atMidHi;
_p8 := NOT gCtrl.main.noFaults;
IF gCtrl.palletDispenser.atMidHi OR NOT gCtrl.main.noFaults THEN
    gCtrl.palletDispenser.hmiBtnClawsLiftToMidHi := FALSE;
END_IF;
IF _p7 OR _p8 THEN gCtrl.palletDispenser.flagClawsLiftToMidHi := FALSE; END_IF;

(* Network 17 *)
_p9 := gCtrl.palletDispenser.atMidLo;
_p10 := NOT gCtrl.main.noFaults;
IF gCtrl.palletDispenser.atMidLo OR NOT gCtrl.main.noFaults THEN
    gCtrl.palletDispenser.hmiBtnClawsLiftToMidLo := FALSE;
END_IF;
IF _p9 OR _p10 THEN gCtrl.palletDispenser.flagClawsLiftToMidLo := FALSE; END_IF;

(* Network 18 *)
IF gCtrl.palletDispenser.atBottom OR NOT gCtrl.main.noFaults THEN
    gCtrl.palletDispenser.hmiBtnClawsLiftToBottom := FALSE;
END_IF;

(* Network 19: ============================================================================ Pallet claws control *)
gMachineIO.dout.PalletClawsClose_SOL7A := gCtrl.main.noFaults AND gCtrl.palletDispenser.hmiBtnPalletClawsOpenClose;

(* Network 20 *)
gMachineIO.dout.PalletClawsOpen_SOL7B := NOT gMachineIO.dout.PalletClawsClose_SOL7A;

(* Network 21 *) (* commented out *)
// IF NOT gCtrl.main.noFaults THEN gMachineIO.dout.PalletClawsClose_SOL7A := FALSE; END_IF;
END_PROGRAM
```

### Program Logical/MachineControl/retainbar

#### Cyclic.ld
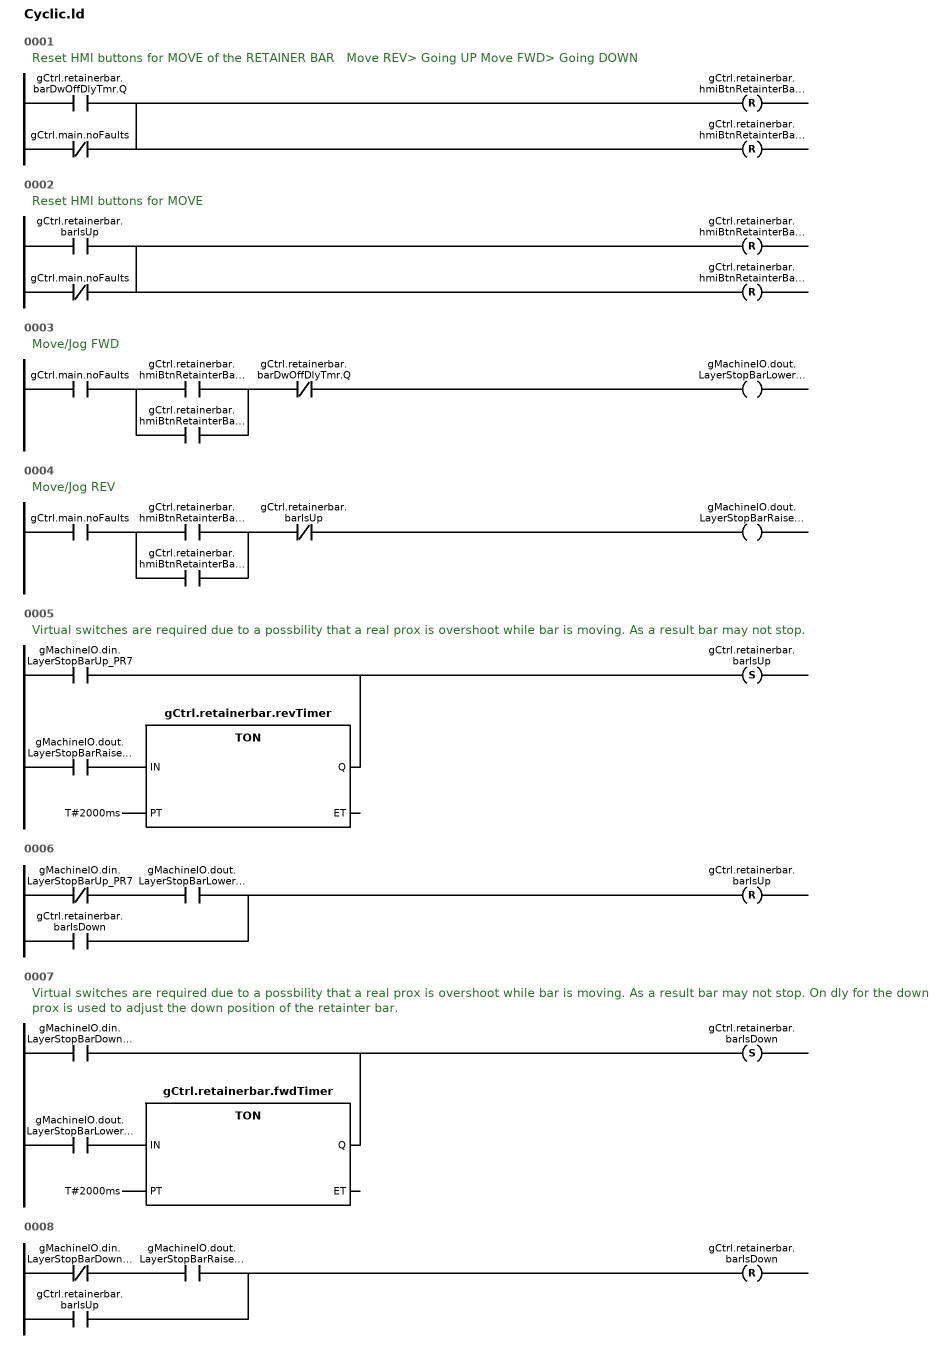
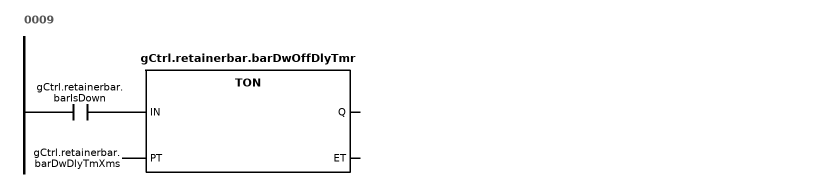
Ladder, written as Structured Text:
```iecst
PROGRAM _CYCLIC
VAR
    _p1 : BOOL;
    _p2 : BOOL;
    _p3 : BOOL;
    _p4 : BOOL;
END_VAR
(* Network 1: Reset HMI buttons for MOVE of the RETAINER BAR   Move REV> Going UP Move FWD> Going DOWN *)
_p1 := gCtrl.retainerbar.barDwOffDlyTmr.Q;
_p2 := NOT gCtrl.main.noFaults;
IF gCtrl.retainerbar.barDwOffDlyTmr.Q OR NOT gCtrl.main.noFaults THEN
    gCtrl.retainerbar.hmiBtnRetainterBarFwd := FALSE;
END_IF;
IF _p1 OR _p2 THEN gCtrl.retainerbar.hmiBtnRetainterBarFwdJog := FALSE; END_IF;

(* Network 2: Reset HMI buttons for MOVE *)
_p3 := gCtrl.retainerbar.barIsUp;
_p4 := NOT gCtrl.main.noFaults;
IF gCtrl.retainerbar.barIsUp OR NOT gCtrl.main.noFaults THEN
    gCtrl.retainerbar.hmiBtnRetainterBarRev := FALSE;
END_IF;
IF _p3 OR _p4 THEN gCtrl.retainerbar.hmiBtnRetainterBarRevJog := FALSE; END_IF;

(* Network 3: Move/Jog FWD *)
gMachineIO.dout.LayerStopBarLower_M3R := gCtrl.main.noFaults AND (gCtrl.retainerbar.hmiBtnRetainterBarFwd OR gCtrl.retainerbar.hmiBtnRetainterBarFwdJog) AND NOT gCtrl.retainerbar.barDwOffDlyTmr.Q;

(* Network 4: Move/Jog REV *)
gMachineIO.dout.LayerStopBarRaise_M3F := gCtrl.main.noFaults AND (gCtrl.retainerbar.hmiBtnRetainterBarRev OR gCtrl.retainerbar.hmiBtnRetainterBarRevJog) AND NOT gCtrl.retainerbar.barIsUp;

(* Network 5: Virtual switches are required due to a possbility that a real prox is overshoot while bar is moving. As a result bar may not stop. *)
IF gMachineIO.din.LayerStopBarUp_PR7 OR gCtrl.retainerbar.revTimer.Q THEN
    gCtrl.retainerbar.barIsUp := TRUE;
END_IF;
gCtrl.retainerbar.revTimer(IN := gMachineIO.dout.LayerStopBarRaise_M3F, PT := T#2000ms);

(* Network 6 *)
IF (NOT gMachineIO.din.LayerStopBarUp_PR7 AND gMachineIO.dout.LayerStopBarLower_M3R) OR gCtrl.retainerbar.barIsDown THEN
    gCtrl.retainerbar.barIsUp := FALSE;
END_IF;

(* Network 7: Virtual switches are required due to a possbility that a real prox is overshoot while bar is moving. As a result bar may not stop. On dly for the down prox is used to adjust the down position of the retainter bar. *)
IF gMachineIO.din.LayerStopBarDown_PR8 OR gCtrl.retainerbar.fwdTimer.Q THEN
    gCtrl.retainerbar.barIsDown := TRUE;
END_IF;
gCtrl.retainerbar.fwdTimer(IN := gMachineIO.dout.LayerStopBarLower_M3R, PT := T#2000ms);

(* Network 8 *)
IF (NOT gMachineIO.din.LayerStopBarDown_PR8 AND gMachineIO.dout.LayerStopBarRaise_M3F) OR gCtrl.retainerbar.barIsUp THEN
    gCtrl.retainerbar.barIsDown := FALSE;
END_IF;

(* Network 9 *)
gCtrl.retainerbar.barDwOffDlyTmr(IN := gCtrl.retainerbar.barIsDown, PT := gCtrl.retainerbar.barDwDlyTmXms);
END_PROGRAM
```

### Program Logical/paiComponents/bglib

#### bgBufMemAlloc.c
```c
#ifndef _BG_BUFMEMALLOC_C
#define _BG_BUFMEMALLOC_C

#include "bgBufMemAlloc.h"
//#include "string.h"

/*
##################################################################################
Buffer memory allocation
##################################################################################
*/
void bgBufMemAllocInit(bgBufMemAlloc_typ* p, char* pBufMem, int lengthBufMemBytes)
{
int i;

	p->pBufMem = pBufMem;
	p->lengthBufMemBytes = lengthBufMemBytes;
	p->lengthUsedMemBytes = 0;
	p->countUsedBlocks = 0;
	p->countMaxBlocks = BGBUFMEMALLOC_MAX_BLOCKS;
	for(i=0; i < p->countMaxBlocks; i++){
		p->memBlock[i].used = 0;
		p->memBlock[i].pMemBlock = 0;
		p->memBlock[i].lengthMemBlockBytes = 0;
	}
}

int bgBufMemAllocCreateBlock(bgBufMemAlloc_typ* p, int blockSize, char** pMemBlock, int* sizeMemBlock)
{
int i;
int availableBufMem = p->lengthBufMemBytes - p->lengthUsedMemBytes;

	if(blockSize >= availableBufMem)
		goto errorExit;

	if(p->countUsedBlocks >= p->countMaxBlocks)
		goto errorExit;

	for(i=0; i < p->countMaxBlocks; i++){
		if(!p->memBlock[i].used){
			p->memBlock[i].used = 1;
			p->memBlock[i].pMemBlock = (p->pBufMem + p->lengthUsedMemBytes);
			/*0 block size - use all available memory*/
			if(!blockSize)
				blockSize = availableBufMem;
			p->memBlock[i].lengthMemBlockBytes = blockSize;
			p->lengthUsedMemBytes += blockSize;
			p->countUsedBlocks++;
			if(pMemBlock)
				*pMemBlock = p->memBlock[i].pMemBlock;
			if(sizeMemBlock)
				*sizeMemBlock = p->memBlock[i].lengthMemBlockBytes;
			return 0;
		}
	}

errorExit:
	if(pMemBlock)
		*pMemBlock = 0;
	if(sizeMemBlock)
		*sizeMemBlock = 0;
	return 1;
}

char* bgBufMemAllocGetBlockPtr(bgBufMemAlloc_typ* p, int blockId, int* blockSize)
{
	if(blockSize)
		*blockSize = 0;

	if((blockId < p->countMaxBlocks) && (!p->memBlock[blockId].used)){
		if(blockSize)
			*blockSize = p->memBlock[blockId].lengthMemBlockBytes;
		return	p->memBlock[blockId].pMemBlock;
	}

	return 0;
}

/*
##################################################################################
String heap
##################################################################################
*/
char* bgStringHeapInit(bgStringHeap_typ* pHeap, char* pHeapMem, int memSize)
{
	pHeap->pMemStart = pHeapMem;
	pHeap->pMemCurrent = pHeap->pMemStart;
	*pHeap->pMemCurrent = 0;
	pHeap->memSize = memSize;
	pHeap->memFree = pHeap->memSize;
	return pHeap->pMemStart;
}

char* bgStringHeapAddString(bgStringHeap_typ* pHeap, char* pStr)
{
int len = strlen(pStr);
char* pCurString = pHeap->pMemCurrent;;

	/*adjust lentgh for 0 termination*/
	len += 1;

	if( len >= pHeap->memFree )
		return 0;

	brsstrcpy((UDINT)pCurString, (UDINT)pStr);

	/*move current ptr*/
	pHeap->pMemCurrent += len;

	/*reduce free mem*/
	pHeap->memFree -= len;

	return pCurString;
}
#endif
```

#### bgHttpProtocol.c
```c
/*
File: bgHttpProtocol.c
=====

*/

/*
B&R components:
===============================================================================
*/
#ifndef WIN32
#include <bur/plc.h>
#include <bur/plctypes.h>
#include <astcp.h>
#include <string.h>
#include <brsystem.h>
#include <sys_lib.h>
#endif

/*
BG components
===============================================================================
*/
#include "bgdebug.h"
#include "bgstring.h"
#include "bgsscanf.h"
#include "bgTcpSocketClientServer.h"
#include "bgHttpProtocol.h"

static void addLine(bgTcpSocketSession_typ* pSession, char* s)
{
char* pDst = (pSession->pSendBuf + pSession->curIdxSendBuf);
int len = strlen(s);

/*
	if( bgHttpSendBufMonitorOverflow(pSession) )
		return;
*/

	brsstrcpy((UDINT)pDst, (UDINT)s);
	pSession->curIdxSendBuf += len;
	brsstrcat((UDINT)pDst,(UDINT) BGHTTP_CONST_STRING_CRLF);
	pSession->curIdxSendBuf += strlen(BGHTTP_CONST_STRING_CRLF);
}

static int bgHttpClientProcessResponse(bgTcpSocketSession_typ* pSession);
static void bgHttpClientSessionAppMemAlloc(bgTcpSocketSession_typ* pSession);
static void bgHttpServerSessionAppMemAlloc(bgTcpSocketSession_typ* pSession);
static void bgHttpSendBufReset(bgTcpSocketSession_typ* pSession);
static void bgHttpSendBufApndHeaderLine(bgTcpSocketSession_typ* pSession, char* headerLine);
static void bgHttpSendBufApndHeaderEnd(bgTcpSocketSession_typ* pSession);
static void bgHttpSendBufApndContentLine(bgTcpSocketSession_typ* pSession, char* contentLine);
static void bgHttpSendBufApndContentEnd(bgTcpSocketSession_typ* pSession);
static int bgHttpSendBufMonitorOverflow(bgTcpSocketSession_typ* pSession, int newLineSize);
static void bgHttpSendBufFillContentSize(bgTcpSocketSession_typ* pSession);
static char* bgHttpGetResponseMsg(int responseCode);
static int bgHttpServerProcessRequest(bgTcpSocketSession_typ* p);
static int bgHttpReceiverGetContentLengthAndPosition(bgTcpSocketSession_typ* pSession);
static int bgHttpReceiver(bgTcpSocketSession_typ* pSession);
static void bgHttpSendBufApndHeaderLineAndFormat(bgTcpSocketSession_typ* pSession, char* headerKeyword, char* value);
static void bgHttpServerSendResponseSetHeader(bgTcpSocketSession_typ* pSession, int responseCode, int contentSize, char* contentType);
static void bgHttpSendBufCallback(bgTcpSocketSession_typ* pSession);
static void bgHttpSendBufDebug(bgTcpSocketSession_typ* pSession);
static void bgHttpRecvBufDebug(bgTcpSocketSession_typ* pSession);

/*
HTTP Protocol
######################################################################################################
######################################################################################################
######################################################################################################
######################################################################################################
*/
void bgHttpServerSessionHandler(bgTcpSocketSession_typ* pSession)
{
	if(pSession->init){
		DBGMSG("bgHttpServerSessionHandler(): init\r\n");
		bgHttpServerSessionAppMemAlloc(pSession);
		/*init receive byte count*/
		pSession->rxByteCount = 0;
		return;
	}

	if( !pSession->initOk ){
		DBGMSG("bgHttpServerSessionHandler(): can't execute session; init NOT OK\r\n");
		return;
	}

	DBGMSG("bgHttpServerSessionHandler(): execute\r\n");

	if( bgHttpReceiver(pSession) )
		return;		/*http receive is NOT complete; continue with receiving*/

	if( pSession->dbgDumpRecvBuf )
		bgHttpRecvBufDebug(pSession);

	if( bgHttpServerProcessRequest(pSession) )
        return;		/*http request error; terminate session*/

    /*http receive success; execute application/protocol layer*/
    {
        bgTcpSocketServer_typ* pServer = (bgTcpSocketServer_typ*)pSession->pTcpLayer;
        if( pServer->pApplicationHandler )
            (*pServer->pApplicationHandler)(pSession);
        else
            bgHttpSendErrorResponse(pSession, 501);
    }
}

void bgHttpServerSendResponse(bgTcpSocketSession_typ* pSession, int responseCode, char* pContent , int contentSize, char* contentType)
{

    	/*init/reset send buffer*/
	bgHttpSendBufReset(pSession);

    /*define HTTP header entries*/
    bgHttpServerSendResponseSetHeader(pSession, responseCode, contentSize, contentType);

	/*append content, if any*/
	if(pContent && contentSize)
		brsstrcat((UDINT)pSession->pSendBuf, (UDINT)pContent);

	pSession->tcpSend.datalen = strlen(pSession->pSendBuf);
	bgHttpSendData(pSession);
	DBGMSG("bgHttpServerSendResponse: rspCode=[%d], totalLen=%d, contentSize=%d\r\n",
     responseCode, pSession->tcpSend.datalen, contentSize);
}

void bgHttpServerSendResponseBeg(bgTcpSocketSession_typ* pSession, int responseCode, char* contentType)
{
    /*init/reset send buffer*/
	bgHttpSendBufReset(pSession);

    /*define HTTP header entries*/
    bgHttpServerSendResponseSetHeader(pSession, responseCode, 1234567, contentType);
	DBGMSG("bgHttpServerSendResponseBeg: rspCode=[%d]\r\n", responseCode);
}

void bgHttpServerSendResponseEnd(bgTcpSocketSession_typ* pSession)
{

	bgHttpSendBufApndContentEnd(pSession);
	bgHttpSendBufFillContentSize(pSession);
	pSession->tcpSend.datalen = strlen(pSession->pSendBuf);
	bgHttpSendData(pSession);
	DBGMSG("bgHttpServerSendResponseEnd: totalLen=%d\r\n", pSession->tcpSend.datalen);
}

static void bgHttpServerSessionAppMemAlloc(bgTcpSocketSession_typ* pSession)
{
/*
 	HTTP session:
 	On init, "alocate" memory within the session application space.

	Session/Application memory allocation:

	-each session/application is given  memory space
	-size of the app space (APPLICATION BUFFER SIZE) is defined in the server init call:
		i.e. bgTcpSocketServerInit(&bgXmlRpcServerData, ... 2048, ...);

	- depending on the application/session needs, this space can be further devided into
	"allocated" memory blocks. See bgBufMemAllocXXX object

	pAppBuffer allocation scheme for bgHttpServerSessionHandler:
		struct httpMessage_typ		--- sizeof(httpMessage_typ) bytes
		listHeaderLines Ptr-s		--- 32 * sizeof(char*) = 128 bytes (holds max 32 items)
		list1 						--- 32 * sizeof(char*) = 128 bytes (holds max 32 items)
		remainig space: listContentLines ptr-s (i.e. 1kBytes of space is 256 items (lines) in the list

*/
char* pMem;
int sizeMem;
httpMessage_typ* pHttpMsg;

	/*set initOk to NOT OK*/
	pSession->initOk = 0;

	bgBufMemAllocInit(&pSession->sessionMem, pSession->pAppBuf, pSession->appBufLength);

	/*1) protocol/application specific data structure, upper layer*/
	if( bgBufMemAllocCreateBlock(&pSession->sessionMem, sizeof(httpMessage_typ) + sizeof(char*), &pMem, &sizeMem) )
	{
    	DBGMSG("bgHttpServerSessionHandler(): init; FATAL ERROR (1); No memory\r\n");
		return;
	}

	pHttpMsg = (httpMessage_typ*)pMem;
	pSession->pProtocol = (char*)pHttpMsg;

	/*2) set storage for list of http header lines (anticipated short list of items)*/
	if( bgBufMemAllocCreateBlock(&pSession->sessionMem, 33 * sizeof(char *), &pMem, &sizeMem) )
	{
    	DBGMSG("bgHttpServerSessionHandler(): init; FATAL ERROR (2); No memory\r\n");
		return;
	}
	bgStringListExMemSet(&pHttpMsg->listHeaderLines, pMem, 32 * sizeof(char *));

	/*3) set storage for short helper list (short list of items, i.e. 32)*/
	if( bgBufMemAllocCreateBlock(&pSession->sessionMem, 33 * sizeof(char *), &pMem, &sizeMem) )
	{
    	DBGMSG("bgHttpServerSessionHandler(): init; FATAL ERROR (3); No memory\r\n");
		return;
	}
    bgStringListExMemSet(&pHttpMsg->list1, pMem, 32 * sizeof(char *));

#if 0
	/*4) set storage for line list (long list of items, i.e. several hundred items, depending on the memory)*/
	if( bgBufMemAllocCreateBlock(&pSession->sessionMem, 0, &pMem, &sizeMem) )
	{
    	DBGMSG("bgHttpServerSessionHandler(): init; FATAL ERROR (4); No memory\r\n");
		return;
	}
    bgStringListExMemSet(&pHttpMsg->listContentLines, pMem, sizeMem);
#endif

	/*init OK*/
	pSession->initOk = 1;

#if 0
	/*dump appliction buffer memory allocation*/
	{
	int i;
	DBGMSG("bgHttpServerSessionHandler: bufMemAlloc total=%d, used=%d, blocks=%d\r\n",
		pSession->sessionMem.lengthBufMemBytes,
		pSession->sessionMem.lengthUsedMemBytes,
		pSession->sessionMem.countUsedBlocks);
	for(i=0; i<pSession->sessionMem.countUsedBlocks; i++){
		DBGMSG("bgHttpServerSessionHandler: bufMemAlloc i=%d, p=%x, l=%d\r\n",
		i,
		pSession->sessionMem.memBlock[i].pMemBlock,
		pSession->sessionMem.memBlock[i].lengthMemBlockBytes);
	}
	}
#endif
}

/*
####################################################################################################
####################################################################################################
####################################################################################################
*/
void bgHttpClientSetConnection(bgTcpSocketClient_typ* pClient, char* serverIpAddr, int serverPortNumber)
{
	if(serverIpAddr)
		brsstrcpy((UDINT)pClient->serverIpAddr, (UDINT)serverIpAddr);

	if(serverPortNumber)
		pClient->serverPort = serverPortNumber;

	DBGMSG("bgHttpClientSetConnection: ip=[%s], port=%d\r\n", serverIpAddr?serverIpAddr:"none", serverPortNumber);

}

void bgHttpClientSendRequest(bgTcpSocketClient_typ* pClient, char* pCmd, char* pContent , int contentSize, char* contentType)
{
bgTcpSocketSession_typ *pSession = &pClient->session[0];

	if( pSession->socketState == BGTCPSOCK_SESSION_STATE_NONE){

        /*init client app specific memory*/
		bgHttpClientSessionAppMemAlloc(pSession);

        /*init/reset send buffer*/
		bgHttpSendBufReset(pSession);

        /*define HTTP header entries*/
        bgHttpClientSendRequestSetHeader(pSession, pCmd, contentSize, contentType);

		/*append content, if any*/
		if(pContent && contentSize)
			brsstrcat((UDINT)pSession->pSendBuf, (UDINT)pContent);

		pSession->tcpSend.datalen = strlen(pSession->pSendBuf);
		bgHttpSendData(pSession);
		DBGMSG("bgHttpClientSendRequest: cmd=[%s], totalLen=%d, contentSize=%d\r\n", pCmd?pCmd:"none", pSession->tcpSend.datalen,contentSize);
	}else{
		DBGMSG("bgHttpClientSendRequest(): rejected! Client is busy!\r\n");
	}
}

void bgHttpClientSessionHandler(bgTcpSocketSession_typ* pSession)
{
	if(pSession->init){
		DBGMSG("bgHttpClientSessionHandler(): init\r\n");
#if 0
NOTE: client memalloc takes place during send request
		bgHttpClientSessionAppMemAlloc(pSession);
#endif
		/*init receive byte count*/
		pSession->rxByteCount = 0;
		return;
	}

	if( !pSession->initOk ){
		DBGMSG("bgHttpClientSessionHandler(): can't execute session; init NOT OK\r\n");
		return;
	}

	DBGMSG("bgHttpClientSessionHandler(): execute\r\n");

	if( bgHttpReceiver(pSession) )
		return;		/*http receive is NOT complete; continue with receiving*/

	DBGMSG("bgHttpClientSessionHandler: recv complete!\r\n");

	if( pSession->dbgDumpRecvBuf )
		bgHttpRecvBufDebug(pSession);

	if( bgHttpClientProcessResponse(pSession) ){
		/*terminate session*/
		DBGMSG("bgHttpClientSessionHandler: http response error\r\n");
		pSession->bCloseSession = 1;
        return;		/*error in http response; terminate session*/
	}

    /*http receive success; execute application/protocol layer*/
    {
        bgTcpSocketClient_typ* pClient = (bgTcpSocketClient_typ*)pSession->pTcpLayer;
        if( pClient->pApplicationHandler )
            (*pClient->pApplicationHandler)(pSession);
        else
			DBGMSG("bgHttpClientSessionHandler: app handler not defined!\r\n");
    }

	/*terminate session*/
	pSession->bCloseSession = 1;
}

static void bgHttpClientSessionAppMemAlloc(bgTcpSocketSession_typ* pSession)
{
/*
 	HTTP session:
 	On init, "alocate" memory within the session application space.

	Session/Application memory allocation:

	-each session/application is given  memory space
	-size of the app space (APPLICATION BUFFER SIZE) is defined in the server init call:
		i.e. bgTcpSocketServerInit(&bgXmlRpcServerData, ... 2048, ...);

	- depending on the application/session needs, this space can be further devided into
	"allocated" memory blocks. See bgBufMemAllocXXX object

	pAppBuffer allocation scheme for bgHttpClientSessionHandler:
		struct httpMessage_typ		--- sizeof(httpMessage_typ) bytes
		listHeaderLines Ptr-s		--- 32 * sizeof(char*) = 128 bytes (holds max 32 items)
		list1 						--- 32 * sizeof(char*) = 128 bytes (holds max 32 items)
		remainig space: listContentLines ptr-s (i.e. 1kBytes of space is 256 items (lines) in the list

*/
httpMessage_typ* pHttpMsg;
char* pMem;
int sizeMem;

    /*simple, session specific memory allocation*/
	pSession->initOk = 0;

	bgBufMemAllocInit(&pSession->sessionMem, pSession->pAppBuf, pSession->appBufLength);

	/*1) protocol/application specific data structure, upper layer*/
	if( bgBufMemAllocCreateBlock(&pSession->sessionMem, sizeof(httpMessage_typ) + sizeof(char*), &pMem, &sizeMem) )
	{
    	DBGMSG("bgHttpClientSessionAppMemAlloc(): FATAL ERROR (1); No memory\r\n");
		return;
	}
	pHttpMsg = (httpMessage_typ*)pMem;
	pSession->pProtocol = (char*)pHttpMsg;

	/*2) set storage for list of http header lines (anticipated short list of items)*/
	if( bgBufMemAllocCreateBlock(&pSession->sessionMem, 33 * sizeof(char *), &pMem, &sizeMem) )
	{
    	DBGMSG("bgHttpClientSessionAppMemAlloc(): FATAL ERROR (2); No memory\r\n");
		return;
	}
	bgStringListExMemSet(&pHttpMsg->listHeaderLines, pMem, 32 * sizeof(char *));

	/*3) set storage for short helper list (short list of items, i.e. 32)*/
	if( bgBufMemAllocCreateBlock(&pSession->sessionMem, 33 * sizeof(char *), &pMem, &sizeMem) )
	{
    	DBGMSG("bgHttpClientSessionAppMemAlloc(): FATAL ERROR (3); No memory\r\n");
		return;
	}
    bgStringListExMemSet(&pHttpMsg->list1, pMem, 32 * sizeof(char *));

	pSession->initOk = 1;

#if 0
	/*dump appliction buffer memory allocation*/
	{
	int i;
	DBGMSG("bgHttpClientSessionHandler: bufMemAlloc total=%d, used=%d, blocks=%d\r\n",
		pSession->sessionMem.lengthBufMemBytes,
		pSession->sessionMem.lengthUsedMemBytes,
		pSession->sessionMem.countUsedBlocks);
	for(i=0; i<pSession->sessionMem.countUsedBlocks; i++){
		DBGMSG("bgHttpClientSessionHandler: bufMemAlloc i=%d, p=%x, l=%d\r\n",
		i,
		pSession->sessionMem.memBlock[i].pMemBlock,
		pSession->sessionMem.memBlock[i].lengthMemBlockBytes);
	}
	}
#endif
}

/*
####################################################################################################
####################################################################################################
####################################################################################################
*/

 int bgHttpReceiver(bgTcpSocketSession_typ* pSession)
{
/*session/application/protocol specific data structure*/
httpMessage_typ* r = (httpMessage_typ*)pSession->pProtocol;
int contentSizeReceived = 0;
int rxInitFlag = pSession->rxByteCount ? 0 : 1;

	DBGMSG("bgHttpReceiver: rxLen=%d, rxInit=%d\r\n", pSession->tcpRecv.recvlen, rxInitFlag);

	/*keep track of bytes received*/
	pSession->rxByteCount += pSession->tcpRecv.recvlen;

	/*http is a character based protocol! always terminate rxBuffer for later string processing*/
	pSession->pRecvBuf[pSession->rxByteCount] = 0;

	/*is this is a first chunk of data recv for this session?*/
	if(rxInitFlag){
		/*check if http content definiton is present in http header;
		if yes, set following values:
		r->contentLength 	is the value extracted from the http header attribute "Content-Length"
		r->contentPosition 	is the offset (position) of the content start within the recvBuf
		*/
		if( !bgHttpReceiverGetContentLengthAndPosition(pSession) ){
			/*header line with "Content-Length" not received; recv complete; next: process request*/
			return 0;
		}

		DBGMSG("bgHttpReceiver: content=YES; contentLength=%d, contentOffset=%d\r\n",
			r->contentLength, r->contentPosition);

		/*check if the entire content is received*/
		if( r->contentPosition > pSession->rxByteCount){
			/*upps! adjust here*/
			DBGMSG("bgHttpReceiver: WARNING conStart=%d > rxLen=%d. Adjusting...\r\n",
			r->contentPosition, pSession->rxByteCount);
			r->contentPosition = pSession->rxByteCount;
		}
	}

	/*monitor if the entire http message is received, including content*/
	contentSizeReceived = pSession->rxByteCount - r->contentPosition;

	/*if received content is less then 2/3 of needed content > continue receiving*/
	if(contentSizeReceived < ((r->contentLength * 2) / 3 )){
		DBGMSG("bgHttpReceiver: incomplete; totalBytesRcvd=%d contentRcvd=%d, contentNeeded=%d\r\n",
			pSession->rxByteCount,
			contentSizeReceived,
			r->contentLength);

		/*continue receiving!*/

		/*adjust parameters of the tcprecv*/
		pSession->tcpRecv.pData = (UDINT)(&pSession->pRecvBuf[pSession->rxByteCount]);	/* address of the buffer */;
		pSession->tcpRecv.datamax = pSession->recvBufLength - pSession->rxByteCount; 	/* length of the buffer */;
		return 1;
	}

	DBGMSG("bgHttpReceiver: Complete; totalBytesRcvd=%d contentRcvd=%d, contentNeeded=%d\r\n",
		pSession->rxByteCount,
		contentSizeReceived,
		r->contentLength);

	return 0;
}

 int bgHttpReceiverGetContentLengthAndPosition(bgTcpSocketSession_typ* pSession)
{
/*session/application/protocol specific data structure*/
httpMessage_typ* r = (httpMessage_typ*)pSession->pProtocol;

int position=0;
int positionHeaderContentLenBegin=0;
int positionHeaderContentLenEnd=0;
char textBuffer[255];

	r->contentLength = 0;
	r->contentPosition = 0;

	/*find if "Content-Length" keyword is present in the request*/
	positionHeaderContentLenBegin = bgStrFindEx(pSession->pRecvBuf, BGHTTP_HEADER_KEY_CONLEN, -1, -1, 1);

	if( positionHeaderContentLenBegin < 0){
		/*content length not present; receive is complete; next: process http request*/
		DBGMSG("bgHttpReceiver: no content\r\n");
		return 0;
	}

	/*content is present! extract the content size & find where it starts!*/
	positionHeaderContentLenEnd = bgStrFindEOL(pSession->pRecvBuf, positionHeaderContentLenBegin);

	/*sanity check*/
	if( (positionHeaderContentLenEnd < 0) ||
		(positionHeaderContentLenEnd >= pSession->rxByteCount) ||
		((positionHeaderContentLenEnd - positionHeaderContentLenBegin) >= 255) ){
		/*can't extract content length; receive is complete; next: process http request*/
		DBGMSG("bgHttpReceiver: can't find end marker\r\n");
		return 0;
	}

	/*extract header line "Content-Length"*/
	bgStrCopyFromTo(pSession->pRecvBuf, positionHeaderContentLenBegin, positionHeaderContentLenEnd, textBuffer);
	/*find value*/
	position = bgStrFind(textBuffer, ":", -1, -1);
	if( position < 0 ){
		/*can't extract content length; receive is complete; next: process http request*/
		DBGMSG("bgHttpReceiver: can't find separator marker [%s]\r\n", textBuffer);
		return 0;
	}
	/*convert received value*/
	bgsscanf(&textBuffer[position+1], "%d", &r->contentLength);
	DBGMSG("bgHttpReceiver: headerLine=[%s], length=%d\r\n", textBuffer, r->contentLength);

	if( !r->contentLength ){
		/*content length not present; receive is complete; next: process http request*/
		DBGMSG("bgHttpReceiver: contentLen=0, process request\r\n");
		return 0;
	}

	/*find content start position within the recvBuf; content comes after header; separation is one empty line!
	*/

	/*positionHeaderContentLenEnd - holds the EOL position for header line "Content-Length". Before the
	seprator (empty) line, there may be more header lines*/
	/*TODO: detect the exact position of the content start!!!*/

	/*Assume that the content start just after the above header line!*/
	r->contentPosition = positionHeaderContentLenEnd + 1;
 	{
		/*search for a first empty line after the content header line -> empty line
		is the separator between the header and the content*/
		int state = 0;
		int idx = r->contentPosition;
		char c;
		while(1){
			c = pSession->pRecvBuf[idx];
			switch(state){
				case 0:
					if( c == '\n' ){
						state = 1;
					}else
					if( c == 0){
						return 1;
					}
					idx++;
				break;
				case 1:
					if( c == '\n' ){
						/*found! two consecutive \n !*/
						r->contentPosition = idx + 1;
						return 1;
					}else
					if( c == '\r'){
						/*ignore \r */
					}else
					if( c == 0){
						return 1;
					}else{
						/*continue searching for the empty line*/
						state = 0;
					}
					idx++;
				break;
			}
		}
	}

}

/*
####################################################################################################
####################################################################################################
####################################################################################################
*/

 int bgHttpServerProcessRequest(bgTcpSocketSession_typ* pSession)
{
/*
This function parses and analyzes standard HTTP request (HTTP/0.9, HTTP/1.0, HTTP1.1).
As a result, it fills-in elemetns in the HTTP protocol data structure (httpMessage_typ)

Following is the typical HTTP/1.1 request:

GET /file1.html HTTP/1.1\r\n                    <-- line 0: HTTP command line
Content-Type: text/html\r\n                     <-- line 1 (optional): HTTP Header, 1st Header Line (if present)
Connection: keep-alive\r\n                      <-- line 2 (optional): HTTP Header, 2nd Header Line (if present) (followed by as many header lines as needed)
\r\n                                            <-- line x (optional): Empty line (Marks separation between HTTPHeader (if present) and HTTP Content (if present)
<head>\r\n                                      <-- line (x+1) (optional): HTTP Content (if present), 1st Content line (if present)
<title>HTTP Content in HTML format</title>\r\n  <-- line (x+2, etc) (optional): Additional HTTP Content lines (if present)
</head>\r\n
<body>\r\n
<h1>My Header 1</h1>\r\n
<p>Simple text in HTML format.\r\n
</body>\r\n
\r\n

This function uses/sets following data (using the above sample request):
pSession->pRecvBuf                              <-- tcp rx buffer; holds the entire HTTP request content

(httpMessage_typ)r = pSession->pProtocol        <-- ptr to the httpMessage structure; structure resides within the pSession->pAppBuf memory area
r->listHeaderLines.itemCount = 3;               <-- http msg header has 3 lines
r->listHeaderLines.items[]                      <-- array of ptrs to each of the 3 lines
r->command = "GET";                             <-- command ptr points to "GET"
r->commandId = BGHTTP_REQUEST_COMMAND_GET;
r->url = "/file1.html"                          <-- url ptr points to "/file1.html"
r->versionString = "HTTP/1.1";
r->version = 11;

*/
httpMessage_typ* r;
int i;
int ret = 1;                                    /*mark request as failure*/

    /*session/application/protocol specific data structure*/
    r = (httpMessage_typ*)pSession->pProtocol;

	/*check if http content is present*/
	if( r->contentLength ){
		/*content is present; separate header and content by inserting 0 (string termination)
		at the end of the http header*/
		if( r->contentPosition && (r->contentPosition < pSession->rxByteCount) )
			pSession->pRecvBuf[r->contentPosition - 1] = 0;
		else{
			DBGMSG("bgHttpServerProcessRequest: WARNING! content data invalid! conLen=%d, conPos=%d, rxLen=%d\r\n",
				r->contentLength, r->contentPosition, pSession->rxByteCount);
			r->contentLength = 0;
			r->contentPosition = 0;
		}
	}

	/*parse 1st part of the request; generate list of header lines*/
	if( bgStringListLinesEx(&r->listHeaderLines, &pSession->pRecvBuf[0], 0, 0) < 0 ){
		DBGMSG("bgHttpServerProcessRequest(): Received header too long! SessionId= %d, len = %d, Error=500\r\n",
			pSession->ident, pSession->rxByteCount);
		bgHttpSendErrorResponse(pSession, 500);
 		return ret;
    }

	/*empty request? it should not be possible, but...*/
	if( r->listHeaderLines.itemCount == 0 ){
		DBGMSG("bgHttpServerProcessRequest(): Invalid request! SessionId= %d, len = %d, Error=400\r\n",
			pSession->ident, pSession->rxByteCount);
		bgHttpSendErrorResponse(pSession, 400);
 		return ret;
	}

#if 0
	DBGMSG("bgHttpServerProcessRequest(): Header (lines=%d):\r\n",
		r->listHeaderLines.itemCount);
	DBGMSG("============================================\r\n");
	for(i=0;i < r->listHeaderLines.itemCount;i++){
		DBGMSG("%s\r\n", r->listHeaderLines.items[i]);
	}
	DBGMSG("============================================\r\n\r\n");
#endif

    /*HTTP REQUEST COMMAND:*/
	/*parse first line of the request*/
	bgStringSplitLineEx(&r->list1, ' ', (char*)r->listHeaderLines.items[0], 0, 0);

	/*one or less words in the first line?*/
	if( (r->list1.itemCount <= 1) || (r->list1.itemCount > 3)){
		DBGMSG("bgHttpServerProcessRequest(): Invalid request! SessionId=%d, len =%d, 1stLnWords=%d  Error=400\r\n",
			pSession->ident, pSession->rxByteCount, r->list1.itemCount);
		bgHttpSendErrorResponse(pSession, 400);
 		return ret;
	}

	/*extract httpVersion & url*/
	r->url = (char*)r->list1.items[1];
	if( r->list1.itemCount == 2){
		DBGMSG("bgHttpServerProcessRequest(): Warning! HTTP request wo. protocol version\r\n");
		r->versionString = "HTTP/0.9";
	}else{
		r->versionString = (char*)r->list1.items[2];
	}

	/*extract http command*/
	if( bgStrFind((char*)r->list1.items[0], "GET", -1, -1) != -1){
		r->command = "GET";
		r->commandId = BGHTTP_REQUEST_COMMAND_GET;
	}else
	if( bgStrFind((char*)r->list1.items[0], "POST", -1, -1) != -1){
		r->command = "POST";
		r->commandId = BGHTTP_REQUEST_COMMAND_POST;
	}else{
		DBGMSG("bgHttpServerProcessRequest(): Invalid command! SessionId=%d, len =%d, Command=[%s] Error=400\r\n",
			pSession->ident, pSession->rxByteCount, r->list1.items[0]);
		bgHttpSendErrorResponse(pSession, 400);
 		return ret;
	}

	DBGMSG("bgHttpServerProcessRequest(): request cmd=[%s] url=[%s] ver=[%s]\r\n",
		r->command, r->url, r->versionString);

	/*mark request as OK!*/
 	ret = 0;

	return ret;
}

static int bgHttpClientProcessResponse(bgTcpSocketSession_typ* pSession)
{
/*
This function parses and analyzes standard HTTP response (HTTP/0.9, HTTP/1.0, HTTP1.1).
As a result, it fills-in elemetns in the HTTP protocol data structure (httpMessage_typ)

Following is the typical HTTP/1.0 response:

HTTP/1.0 200 OK\r\n                    			<-- line 0: HTTP response line
Server: SimpleHTTP/0.6 Python/2.5c2				<-- line 1 (optional): HTTP Header, 1st Header Line (if present)
Date: Mon, 23 Jul 2007 02:26:25 GMT				<-- line 2 (optional): HTTP Header, 2nd Header Line (if present)
Content-Type: text/html\r\n                     <-- line 3 (optional): HTTP Header, 3rd Header Line (if present)
\r\n                                            <-- line x (optional): Empty line (Marks separation between HTTPHeader (if present) and HTTP Content (if present)
<head>\r\n                                      <-- line (x+1) (optional): HTTP Content (if present), 1st Content line (if present)
<title>HTTP Content in HTML format</title>\r\n  <-- line (x+2, etc) (optional): Additional HTTP Content lines (if present)
</head>\r\n
<body>\r\n
<h1>My Header 1</h1>\r\n
<p>Simple text in HTML format.\r\n
</body>\r\n
\r\n

This function uses/sets following data (using the above sample request):
pSession->pRecvBuf                              <-- tcp rx buffer; holds the entire HTTP request content

(httpMessage_typ)r = pSession->pProtocol        <-- ptr to the httpMessage structure; structure resides within the pSession->pAppBuf memory area
r->listHeaderLines.itemCount = 3;               <-- response header has 3 lines
r->listHeaderLines.items[]                      <-- array of ptrs to each of the 3 lines
r->command = "OK";                             	<-- command ptr points to "OK" (long response result)
r->commandId = 200;								<-- commandId contains error value, 200
r->versionString = "HTTP/1.0";
r->version = 10;

*/
httpMessage_typ* r;
int i;
int ret = 1;                                    /*mark request as failure*/

    /*session/application/protocol specific data structure*/
    r = (httpMessage_typ*)pSession->pProtocol;

	/*check if http content is present*/
	if( r->contentLength ){
		/*content is present; separate header and content by inserting 0 (string termination)
		at the end of the http header*/
		if( r->contentPosition && (r->contentPosition < pSession->rxByteCount) )
			pSession->pRecvBuf[r->contentPosition - 1] = 0;
		else{
			DBGMSG("bgHttpServerProcessRequest: WARNING! content data invalid! conLen=%d, conPos=%d, rxLen=%d\r\n",
				r->contentLength, r->contentPosition, pSession->rxByteCount);
			r->contentLength = 0;
			r->contentPosition = 0;
		}
	}

	/*parse 1st part of the response; generate list of header lines*/
	if( bgStringListLinesEx(&r->listHeaderLines, &pSession->pRecvBuf[0], 0, 0) < 0 ){
		DBGMSG("bgHttpClientProcessResponse: Received header too long! SessionId= %d, len = %d, Error=500\r\n",
			pSession->ident, pSession->rxByteCount);
 		return ret;
    }

	/*empty request? it should not be possible, but...*/
	if( r->listHeaderLines.itemCount == 0 ){
		DBGMSG("bgHttpClientProcessResponse(): Invalid response! SessionId= %d, len = %d, Error=400\r\n",
			pSession->ident, pSession->rxByteCount);
 		return ret;
	}

#if 0
	DBGMSG("bgHttpClientProcessResponse(): Header (lines=%d):\r\n",
		r->listHeaderLines.itemCount);
	DBGMSG("============================================\r\n");
	for(i=0;i < r->listHeaderLines.itemCount;i++){
		DBGMSG("%s\r\n", r->listHeaderLines.items[i]);
	}
	DBGMSG("============================================\r\n\r\n");
#endif

    /*HTTP RESPONSE:*/
	/*parse first line of the response*/
	bgStringSplitLineEx(&r->list1, ' ', (char*)r->listHeaderLines.items[0], 0, 0);

	/*one or less words in the first line?*/
	if( (r->list1.itemCount <= 1) || (r->list1.itemCount > 3)){
		DBGMSG("bgHttpClientProcessResponse(): Invalid response! SessionId=%d, len =%d, 1stLnWords=%d  Error=400\r\n",
			pSession->ident, pSession->rxByteCount, r->list1.itemCount);
 		return ret;
	}

	/*extract data from the 1st line in response*/
	r->versionString = (char*)r->list1.items[0];
	bgsscanf((char*)r->list1.items[1], "%d", &r->commandId);
	r->command = (char*)r->list1.items[2];

	DBGMSG("bgHttpClientProcessResponse(): response ver=[%s] err=[%d] msg=[%s]\r\n",
		r->versionString, r->commandId, r->command);

	/*mark response as OK!*/
 	ret = 0;

 	return ret;
}

/*
####################################################################################################
####################################################################################################
####################################################################################################
*/
static void bgHttpSendBufReset(bgTcpSocketSession_typ* pSession)
{
/*session/application/protocol specific data structure*/
httpMessage_typ* r = (httpMessage_typ*)pSession->pProtocol;
char* pDst = pSession->pSendBuf;

	/*clr send buffer*/
	*pDst = 0;

	/*reset current ptr into the send buffer; prepare for incremental write*/
	pSession->curIdxSendBuf = 0;

	/*reset length of sections within the send buffer*/
	r->sendHeaderLength = 0;
	r->sendContentLength = 0;
	r->sendTotalLength = 0;
}

static void bgHttpSendBufApndHeaderEnd(bgTcpSocketSession_typ* pSession)
{
/*session/application/protocol specific data structure*/
httpMessage_typ* r = (httpMessage_typ*)pSession->pProtocol;

	addLine(pSession,"");
	r->sendTotalLength = strlen(pSession->pSendBuf);
	r->sendHeaderLength = r->sendTotalLength;
}

static void bgHttpSendBufApndHeaderLine(bgTcpSocketSession_typ* pSession, char* headerLine)
{
	addLine(pSession, headerLine);
}

static void bgHttpSendBufApndHeaderLineAndFormat(bgTcpSocketSession_typ* pSession, char* headerKeyword, char* value)
{
char txt[255];
    bgsprintf(txt, "%s: %s", headerKeyword, value);
	addLine(pSession, txt);
}

static void bgHttpSendBufApndContentLine(bgTcpSocketSession_typ* pSession, char* contentLine)
{
	addLine(pSession, contentLine);
}

static int bgHttpSendBufMonitorOverflow(bgTcpSocketSession_typ* pSession, int newLineSize)
{
 /*as content may be very long, monitor for send buffer overflow!*/
httpMessage_typ* r = (httpMessage_typ*)pSession->pProtocol;

int sendBufTotalSize = pSession->sendBufLength;
int sendBuffUsedSize = r->sendTotalLength;

	if(sendBufTotalSize <= (sendBuffUsedSize + newLineSize + 10)){
		/*trigger error in  bgXXXApplication() (i.e. bgWebServerApplication() )*/
		r->sendTotalLength = pSession->sendBufLength;
		return 1;
	}

	return 0;
}

static void bgHttpSendBufApndContentEnd(bgTcpSocketSession_typ* pSession)
{
httpMessage_typ* r = (httpMessage_typ*)pSession->pProtocol;

	addLine(pSession, "");

	r->sendContentLength = strlen(pSession->pSendBuf) - r->sendHeaderLength;

	bgHttpSendBufFillContentSize(pSession);
}

static void bgHttpSendBufFillContentSize(bgTcpSocketSession_typ* pSession)
{
/*session/application/protocol specific data structure*/
httpMessage_typ* r = (httpMessage_typ*)pSession->pProtocol;
char* pDst = pSession->pSendBuf;
int headerEnd = r->sendHeaderLength;
int lineStart = 0;
int lineEnd = 0;
int separatorStart = 0;
int i;
char txtBuf[32];
/*
This function searches trough the header section of the reply (send) buffer.
When it finds keyword "Content-Length" it sets the value part correctly
(i.e. "Content-Length: 342")
*/

	/*search for keyword within the reply header*/
	lineStart = bgStrFind(pDst, BGHTTP_HEADER_KEY_CONLEN,
		0,
		headerEnd);

	if( lineStart < 0){
		DBGCRT("bgHttpSendBufFillContentSize(): can't find keyword %s\r\n", BGHTTP_HEADER_KEY_CONLEN);
		return;
	}

	/*search for key / value separator*/
	separatorStart = bgStrFind(pDst, ":",
		lineStart,
		headerEnd);

	if( separatorStart < 0){
		DBGCRT("bgHttpSendBufFillContentSize(): can't find separator\r\n");
		return;
	}

	/*search for end of the line with the above keyword*/
	lineEnd = bgStrFind(pDst, BGHTTP_CONST_STRING_CRLF,
		separatorStart,
		headerEnd);

	if( lineEnd < 0){
		DBGCRT("bgHttpSendBufFillContentSize(): can't find EOL\r\n");
		return;
	}

	/*DBGMSG("headerStart=%d, headerEnd=%d, lineStart=%d, sepStart=%d, lineEnd=%d\r\n", headerStart, headerEnd, lineStart, separatorStart, lineEnd);*/

	/*erase existing value by filling spaces*/
	for(i=(separatorStart + 1); i<lineEnd; i++){
		pDst[i] = ' ';
	}

	/*write new value*/
	bgsprintf(&txtBuf[0], "%d", r->sendContentLength);
	memcpy(&pDst[separatorStart + 2], &txtBuf[0], strlen(&txtBuf[0]));

}

void bgHttpSendErrorResponse(bgTcpSocketSession_typ* pSession, int responseCode)
{
/*
Example of error response:

HTTP/1.0 404 Resource Not Found
Server: bgHTTPServer/0.50
Connection: close
Content-Type: text/html
Content-Length: 123

<head>
<title>Error response</title>
</head>
<body>
<h1>Error response</h1>
<p>Error code 404
<p>Message: Resource Not Found.
</body>
*/
char textBuffer[255];

	bgHttpServerSendResponseBeg(pSession, responseCode, "text/html");

	addLine(pSession,"<head>" );
	addLine(pSession,"<title>Error response</title>");
	addLine(pSession,"</head>");
	addLine(pSession,"<body>");
	addLine(pSession,"<h1>Error response</h1>");

	bgsprintf(textBuffer, "<p>Error code %d.", responseCode);
	addLine(pSession,textBuffer);

	bgsprintf(textBuffer, "<p>Message: %s.", bgHttpGetResponseMsg(responseCode) );
	addLine(pSession,textBuffer);

	addLine(pSession,"</body>");

	bgHttpServerSendResponseEnd(pSession);
}

 char* bgHttpGetResponseMsg(int responseCode)
{

	switch(responseCode){
		case 200: return "OK"; break;
		case 400: return "Bad Request"; break;
		case 401: return "Unauthorized"; break;
		case 403: return "Forbidden"; break;
		case 404: return "Resource Not Found"; break;
		case 405: return "Method Not Allowed"; break;
		case 413: return "Requested Entity Too Large"; break;
		case 500: return "Internal Server Error"; break;
		case 501: return "Not Implemented"; break;
		case 505: return "HTTP Version Not Supported"; break;
		default: return "unknown error"; break;
	}
}

void bgHttpClientSendRequestSetHeader(bgTcpSocketSession_typ* pSession, char* pCmd, int contentSize, char* contentType)
{
char txtBuf[255];

    bgsprintf(txtBuf, "%s %s", pCmd, BGHTTP_CONST_STRING_VERSION);
	bgHttpSendBufApndHeaderLine(pSession, txtBuf);

	bgHttpSendBufApndHeaderLine(pSession, "Connection: close");

    if(contentType){
		bgsprintf(txtBuf, "Content-Type: %s", contentType);
		bgHttpSendBufApndHeaderLine(pSession, txtBuf);
}
    else
		bgHttpSendBufApndHeaderLine(pSession, "Content-Type: text/html");

	bgsprintf(txtBuf, "%s: %d", BGHTTP_HEADER_KEY_CONLEN, contentSize);
	bgHttpSendBufApndHeaderLine(pSession, txtBuf);

    /*append empty line - separates header from content & calculate header size*/
	bgHttpSendBufApndHeaderEnd(pSession);
}

static void bgHttpServerSendResponseSetHeader(bgTcpSocketSession_typ* pSession, int responseCode, int contentSize, char* contentType)
{
char txtBuf[255];

    bgsprintf(txtBuf, "%s %d %s", BGHTTP_CONST_STRING_VERSION, responseCode, bgHttpGetResponseMsg(responseCode));
	bgHttpSendBufApndHeaderLine(pSession, txtBuf);

	bgHttpSendBufApndHeaderLine(pSession, "Connection: close");

    if(contentType){
		bgsprintf(txtBuf, "Content-Type: %s", contentType);
		bgHttpSendBufApndHeaderLine(pSession, txtBuf);
}
    else
		bgHttpSendBufApndHeaderLine(pSession, "Content-Type: text/html");

	bgsprintf(txtBuf, "%s: %d", BGHTTP_HEADER_KEY_CONLEN, contentSize);
	bgHttpSendBufApndHeaderLine(pSession, txtBuf);

    /*append empty line - separates header from content & calculate header size*/
    bgHttpSendBufApndHeaderEnd(pSession);
}

void bgHttpSendData(bgTcpSocketSession_typ* pSession)
{
httpMessage_typ* r = (httpMessage_typ*)pSession->pProtocol;
int len = strlen(pSession->pSendBuf);

	if( len !=  r->sendTotalLength){
		DBGMSG("bgTcpSocketServerSessionSendData: Warning! l=%d, t=%d\r\n", len, r->sendTotalLength);
	}

	pSession->txByteCountTotal = len;
	pSession->txByteCount = 0;

	pSession->pSendBufHandler = bgHttpSendBufCallback;

	/*set flag for session layer to send data*/
	pSession->bSendData = 1;

	if(pSession->dbgDumpSendBuf)
		bgHttpSendBufDebug(pSession);
}

static void bgHttpSendBufCallback(bgTcpSocketSession_typ* pSession)
{
	/*incomplete data send*/
	pSession->txByteCount += pSession->tcpSend.sentlen;

	/*adjust send ptr & len*/
	pSession->tcpSend.pData = (UDINT)(&pSession->pSendBuf[pSession->txByteCount]);

	if(pSession->txByteCountTotal > pSession->txByteCount)
		pSession->tcpSend.datalen = pSession->txByteCountTotal - pSession->txByteCount;

}

/*
Dump send buffer.
*/
static void bgHttpSendBufDebug(bgTcpSocketSession_typ* pSession)
{
int i;
int j;
int crFound;
char text[90];
int len = pSession->txByteCountTotal;

	DBGMSG("bgHttpSendBuf dump:(%d bytes)\r\n", len);
	DBGMSG("=================================================================\r\n");
	crFound = 0;
	for(i=0, j=0; i<len; i++){
		text[j] = pSession->pSendBuf[i];

		if( text[j] == '\r' ){
			crFound = 1;
		}

		if( text[j] == '\n'){
			if(!crFound || (crFound > 2) ){
				j++;
				text[j] = '\r';
			}
			crFound = 0;
		}

		if( (j >= 80) || (i >= (len - 1) ) ){
			text[j+1] = 0;
			j = 0;
			DBGMSG("%s", &text[0]);
		}else{
			j++;
		}

		if( crFound )
			crFound++;

	}
	DBGMSG("\r\n=================================================================\r\n");
}

/*
Dump recv buffer.
*/
static void bgHttpRecvBufDebug(bgTcpSocketSession_typ* pSession)
{
int i;
int j;
int crFound;
char text[90];
int len = pSession->rxByteCount;

	DBGMSG("bgHttpRecvBuf dump: (%d bytes)\r\n", len);
	DBGMSG("=================================================================\r\n");
	crFound = 0;
	for(i=0, j=0;i<len; i++){
		text[j] = pSession->pRecvBuf[i];

		if( text[j] == '\r' ){
			crFound = 1;
		}

		if( text[j] == '\n'){
			if(!crFound || (crFound > 2) ){
				j++;
				text[j] = '\r';
			}
			crFound = 0;
		}

		if( (j >= 80) || (i >= (len - 1) ) ){
			text[j+1] = 0;
			j = 0;
			DBGMSG("%s", &text[0]);
		}else{
			j++;
		}

		if( crFound )
			crFound++;

	}
	DBGMSG("\r\n=================================================================\r\n");
}

char* bgHttpGetContentStartAddr(bgTcpSocketSession_typ* pSession)
{
	/*session/application/protocol specific data structure*/
	httpMessage_typ* r = (httpMessage_typ*)pSession->pProtocol;

	return &pSession->pRecvBuf[r->contentPosition];
}
int bgHttpGetContentLength(bgTcpSocketSession_typ* pSession)
{
	/*session/application/protocol specific data structure*/
	httpMessage_typ* r = (httpMessage_typ*)pSession->pProtocol;

	return r->contentLength;
}
```
